gfCNCPoint4[6055] = {X 82.2391, Y 48.2324, Z -5.5000, A 0.000, B 0.000, C 0.000 }
gfCNCPoint4[6056] = {X 81.7221, Y 47.5300, Z -5.5000, A 0.000, B 0.000, C 0.000 }
gfCNCPoint4[6057] = {X 81.3384, Y 46.7467, Z -5.5000, A 0.000, B 0.000, C 0.000 }
gfCNCPoint4[6058] = {X 81.1002, Y 45.9077, Z -5.5000, A 0.000, B 0.000, C 0.000 }
gfCNCPoint4[6059] = {X 81.0152, Y 45.0397, Z -5.5000, A 0.000, B 0.000, C 0.000 }
gfCNCPoint4[6060] = {X 81.0151, Y 44.2040, Z -5.5000, A 0.000, B 0.000, C 0.000 }
gfCNCPoint4[6061] = {X 81.1197, Y 43.2202, Z -5.5000, A 0.000, B 0.000, C 0.000 }
gfCNCPoint4[6062] = {X 81.4183, Y 42.2769, Z -5.5000, A 0.000, B 0.000, C 0.000 }
gfCNCPoint4[6063] = {X 81.8990, Y 41.4122, Z -5.5000, A 0.000, B 0.000, C 0.000 }
gfCNCPoint4[6064] = {X 82.5425, Y 40.6607, Z -5.5000, A 0.000, B 0.000, C 0.000 }
gfCNCPoint4[6065] = {X 82.5423, Y 25.2486, Z -5.5000, A 0.000, B 0.000, C 0.000 }
gfCNCPoint4[6066] = {X 77.7423, Y 25.2486, Z -5.5000, A 0.000, B 0.000, C 0.000 }
gfCNCPoint4[6067] = {X 77.7422, Y 18.1966, Z -5.5000, A 0.000, B 0.000, C 0.000 }
gfCNCPoint4[6068] = {X 77.0779, Y 16.9730, Z -5.5000, A 0.000, B 0.000, C 0.000 }
gfCNCPoint4[6069] = {X 76.5960, Y 15.6668, Z -5.5000, A 0.000, B 0.000, C 0.000 }
gfCNCPoint4[6070] = {X 76.3064, Y 14.3049, Z -5.5000, A 0.000, B 0.000, C 0.000 }
gfCNCPoint4[6071] = {X 74.0412, Y 14.3049, Z -5.5000, A 0.000, B 0.000, C 0.000 }
gfCNCPoint4[6072] = {X 73.9993, Y 14.7005, Z -5.5000, A 0.000, B 0.000, C 0.000 }
gfCNCPoint4[6073] = {X 73.9466, Y 15.0949, Z -5.5000, A 0.000, B 0.000, C 0.000 }
gfCNCPoint4[6074] = {X 77.7423, Y 25.2486, Z -5.5000, A 0.000, B 0.000, C 0.000 }
gfCNCPoint4[6075] = {X 80.1423, Y 25.2486, Z -5.5000, A 0.000, B 0.000, C 0.000 }
gfCNCPoint4[6076] = {X 80.1422, Y 17.4393, Z -5.5000, A 0.000, B 0.000, C 0.000 }
gfCNCPoint4[6077] = {X 79.4941, Y 16.4459, Z -5.5000, A 0.000, B 0.000, C 0.000 }
gfCNCPoint4[6078] = {X 79.0159, Y 15.3604, Z -5.5000, A 0.000, B 0.000, C 0.000 }
gfCNCPoint4[6079] = {X 78.7203, Y 14.2116, Z -5.5000, A 0.000, B 0.000, C 0.000 }
gfCNCPoint4[6080] = {X 78.6153, Y 13.0301, Z -5.5000, A 0.000, B 0.000, C 0.000 }
gfCNCPoint4[6081] = {X 78.6151, Y 12.1868, Z -5.5000, A 0.000, B 0.000, C 0.000 }
gfCNCPoint4[6082] = {X 78.6164, Y 12.0458, Z -5.5000, A 0.000, B 0.000, C 0.000 }
gfCNCPoint4[6083] = {X 78.6205, Y 11.9049, Z -5.5000, A 0.000, B 0.000, C 0.000 }
gfCNCPoint4[6084] = {X 71.6988, Y 11.9049, Z -5.5000, A 0.000, B 0.000, C 0.000 }
gfCNCPoint4[6085] = {X 71.7013, Y 12.0459, Z -5.5000, A 0.000, B 0.000, C 0.000 }
gfCNCPoint4[6086] = {X 71.7021, Y 12.1868, Z -5.5000, A 0.000, B 0.000, C 0.000 }
gfCNCPoint4[6087] = {X 71.7016, Y 13.0911, Z -5.5000, A 0.000, B 0.000, C 0.000 }
gfCNCPoint4[6088] = {X 71.6386, Y 14.2148, Z -5.5000, A 0.000, B 0.000, C 0.000 }
gfCNCPoint4[6089] = {X 71.4714, Y 15.3277, Z -5.5000, A 0.000, B 0.000, C 0.000 }
gfCNCPoint4[6090] = {X 78.9558, Y 35.3487, Z -5.5000, A 0.000, B 0.000, C 0.000 }
gfCNCPoint4[6091] = {X 79.5720, Y 35.9625, Z -5.5000, A 0.000, B 0.000, C 0.000 }
gfCNCPoint4[6092] = {X 80.1424, Y 36.6190, Z -5.5000, A 0.000, B 0.000, C 0.000 }
gfCNCPoint4[6093] = {X 80.1423, Y 25.2486, Z -5.5000, A 0.000, B 0.000, C 0.000 }
gfCNCPoint4[6094] = {X 82.5423, Y 25.2486, Z -5.5000, A 0.000, B 0.000, C 0.000 }
gfCNCPoint4[6095] = {X 82.5422, Y 16.5238, Z -5.5000, A 0.000, B 0.000, C 0.000 }
gfCNCPoint4[6096] = {X 81.9012, Y 15.7822, Z -5.5000, A 0.000, B 0.000, C 0.000 }
gfCNCPoint4[6097] = {X 81.4214, Y 14.9274, Z -5.5000, A 0.000, B 0.000, C 0.000 }
gfCNCPoint4[6098] = {X 81.1220, Y 13.9940, Z -5.5000, A 0.000, B 0.000, C 0.000 }
gfCNCPoint4[6099] = {X 81.0153, Y 13.0196, Z -5.5000, A 0.000, B 0.000, C 0.000 }
gfCNCPoint4[6100] = {X 81.0151, Y 12.1868, Z -5.5000, A 0.000, B 0.000, C 0.000 }
gfCNCPoint4[6101] = {X 81.0160, Y 12.0923, Z -5.5000, A 0.000, B 0.000, C 0.000 }
gfCNCPoint4[6102] = {X 81.0187, Y 11.9979, Z -5.5000, A 0.000, B 0.000, C 0.000 }
gfCNCPoint4[6103] = {X 81.1324, Y 11.1230, Z -5.5000, A 0.000, B 0.000, C 0.000 }
gfCNCPoint4[6104] = {X 81.4018, Y 10.2828, Z -5.5000, A 0.000, B 0.000, C 0.000 }
gfCNCPoint4[6105] = {X 81.8181, Y 9.5049, Z -5.5000, A 0.000, B 0.000, C 0.000 }
gfCNCPoint4[6106] = {X 82.2191, Y 9.7687, Z -5.5000, A 0.000, B 0.000, C 0.000 }
gfCNCPoint4[6107] = {X 82.7659, Y 9.0935, Z -5.5000, A 0.000, B 0.000, C 0.000 }
gfCNCPoint4[6108] = {X 83.4348, Y 8.5389, Z -5.5000, A 0.000, B 0.000, C 0.000 }
gfCNCPoint4[6109] = {X 84.1996, Y 8.1266, Z -5.5000, A 0.000, B 0.000, C 0.000 }
gfCNCPoint4[6110] = {X 85.0305, Y 7.8726, Z -5.5000, A 0.000, B 0.000, C 0.000 }
gfCNCPoint4[6111] = {X 85.8951, Y 7.7868, Z -5.5000, A 0.000, B 0.000, C 0.000 }
gfCNCPoint4[6112] = {X 94.0497, Y 7.7868, Z -5.5000, A 0.000, B 0.000, C 0.000 }
gfCNCPoint4[6113] = {X 95.0288, Y 7.8971, Z -5.5000, A 0.000, B 0.000, C 0.000 }
gfCNCPoint4[6114] = {X 95.9588, Y 8.2226, Z -5.5000, A 0.000, B 0.000, C 0.000 }
gfCNCPoint4[6115] = {X 96.7930, Y 8.7468, Z -5.5000, A 0.000, B 0.000, C 0.000 }
gfCNCPoint4[6116] = {X 97.4897, Y 9.4435, Z -5.5000, A 0.000, B 0.000, C 0.000 }
gfCNCPoint4[6117] = {X 98.0139, Y 10.2777, Z -5.5000, A 0.000, B 0.000, C 0.000 }
gfCNCPoint4[6118] = {X 98.3394, Y 11.2077, Z -5.5000, A 0.000, B 0.000, C 0.000 }
gfCNCPoint4[6119] = {X 98.4497, Y 12.1868, Z -5.5000, A 0.000, B 0.000, C 0.000 }
gfCNCPoint4[6120] = {X 98.4494, Y 13.0233, Z -5.5000, A 0.000, B 0.000, C 0.000 }
gfCNCPoint4[6121] = {X 98.3724, Y 13.7990, Z -5.5000, A 0.000, B 0.000, C 0.000 }
gfCNCPoint4[6122] = {X 98.1597, Y 14.5489, Z -5.5000, A 0.000, B 0.000, C 0.000 }
gfCNCPoint4[6123] = {X 97.8180, Y 15.2496, Z -5.5000, A 0.000, B 0.000, C 0.000 }
gfCNCPoint4[6124] = {X 98.3682, Y 16.6194, Z -5.5000, A 0.000, B 0.000, C 0.000 }
gfCNCPoint4[6125] = {X 101.8748, Y 25.3115, Z -5.5000, A 0.000, B 0.000, C 0.000 }
gfCNCPoint4[6126] = {X 103.4202, Y 21.4659, Z -5.5000, A 0.000, B 0.000, C 0.000 }
gfCNCPoint4[6127] = {X 105.9238, Y 15.2225, Z -5.5000, A 0.000, B 0.000, C 0.000 }
gfCNCPoint4[6128] = {X 105.5855, Y 14.5151, Z -5.5000, A 0.000, B 0.000, C 0.000 }
gfCNCPoint4[6129] = {X 105.3781, Y 13.7589, Z -5.5000, A 0.000, B 0.000, C 0.000 }
gfCNCPoint4[6130] = {X 105.3083, Y 12.9779, Z -5.5000, A 0.000, B 0.000, C 0.000 }
gfCNCPoint4[6131] = {X 105.3083, Y 12.1868, Z -5.5000, A 0.000, B 0.000, C 0.000 }
gfCNCPoint4[6132] = {X 105.4186, Y 11.2077, Z -5.5000, A 0.000, B 0.000, C 0.000 }
gfCNCPoint4[6133] = {X 105.7440, Y 10.2777, Z -5.5000, A 0.000, B 0.000, C 0.000 }
gfCNCPoint4[6134] = {X 106.2682, Y 9.4435, Z -5.5000, A 0.000, B 0.000, C 0.000 }
gfCNCPoint4[6135] = {X 106.9649, Y 8.7468, Z -5.5000, A 0.000, B 0.000, C 0.000 }
gfCNCPoint4[6136] = {X 107.7992, Y 8.2226, Z -5.5000, A 0.000, B 0.000, C 0.000 }
gfCNCPoint4[6137] = {X 108.7292, Y 7.8971, Z -5.5000, A 0.000, B 0.000, C 0.000 }
gfCNCPoint4[6138] = {X 109.7083, Y 7.7868, Z -5.5000, A 0.000, B 0.000, C 0.000 }
gfCNCPoint4[6139] = {X 117.7916, Y 7.7868, Z -5.5000, A 0.000, B 0.000, C 0.000 }
gfCNCPoint4[6140] = {X 118.7707, Y 7.8971, Z -5.5000, A 0.000, B 0.000, C 0.000 }
gfCNCPoint4[6141] = {X 119.7007, Y 8.2226, Z -5.5000, A 0.000, B 0.000, C 0.000 }
gfCNCPoint4[6142] = {X 120.5349, Y 8.7468, Z -5.5000, A 0.000, B 0.000, C 0.000 }
gfCNCPoint4[6143] = {X 121.2316, Y 9.4435, Z -5.5000, A 0.000, B 0.000, C 0.000 }
gfCNCPoint4[6144] = {X 121.7558, Y 10.2777, Z -5.5000, A 0.000, B 0.000, C 0.000 }
gfCNCPoint4[6145] = {X 122.0813, Y 11.2077, Z -5.5000, A 0.000, B 0.000, C 0.000 }
gfCNCPoint4[6146] = {X 122.1916, Y 12.1868, Z -5.5000, A 0.000, B 0.000, C 0.000 }
gfCNCPoint4[6147] = {X 122.1913, Y 13.0233, Z -5.5000, A 0.000, B 0.000, C 0.000 }
gfCNCPoint4[6148] = {X 122.0831, Y 13.9490, Z -5.5000, A 0.000, B 0.000, C 0.000 }
gfCNCPoint4[6149] = {X 121.7823, Y 14.8311, Z -5.5000, A 0.000, B 0.000, C 0.000 }
gfCNCPoint4[6150] = {X 121.3025, Y 15.6301, Z -5.5000, A 0.000, B 0.000, C 0.000 }
gfCNCPoint4[6151] = {X 120.6651, Y 16.3101, Z -5.5000, A 0.000, B 0.000, C 0.000 }
gfCNCPoint4[6152] = {X 120.6644, Y 40.8765, Z -5.5000, A 0.000, B 0.000, C 0.000 }
gfCNCPoint4[6153] = {X 120.6784, Y 40.8882, Z -5.5000, A 0.000, B 0.000, C 0.000 }
gfCNCPoint4[6154] = {X 121.3172, Y 41.5763, Z -5.5000, A 0.000, B 0.000, C 0.000 }
gfCNCPoint4[6155] = {X 121.7955, Y 42.3843, Z -5.5000, A 0.000, B 0.000, C 0.000 }
gfCNCPoint4[6156] = {X 122.0914, Y 43.2753, Z -5.5000, A 0.000, B 0.000, C 0.000 }
gfCNCPoint4[6157] = {X 122.1916, Y 44.2089, Z -5.5000, A 0.000, B 0.000, C 0.000 }
gfCNCPoint4[6158] = {X 122.1916, Y 45.0000, Z -5.5000, A 0.000, B 0.000, C 0.000 }
gfCNCPoint4[6159] = {X 122.0813, Y 45.9791, Z -5.5000, A 0.000, B 0.000, C 0.000 }
gfCNCPoint4[6160] = {X 121.7558, Y 46.9091, Z -5.5000, A 0.000, B 0.000, C 0.000 }
gfCNCPoint4[6161] = {X 121.2316, Y 47.7434, Z -5.5000, A 0.000, B 0.000, C 0.000 }
gfCNCPoint4[6162] = {X 120.5349, Y 48.4401, Z -5.5000, A 0.000, B 0.000, C 0.000 }
gfCNCPoint4[6163] = {X 119.7007, Y 48.9643, Z -5.5000, A 0.000, B 0.000, C 0.000 }
gfCNCPoint4[6164] = {X 118.7707, Y 49.2897, Z -5.5000, A 0.000, B 0.000, C 0.000 }
gfCNCPoint4[6165] = {X 117.7916, Y 49.4000, Z -5.5000, A 0.000, B 0.000, C 0.000 }
gfCNCPoint4[6166] = {X 111.9185, Y 49.4000, Z -5.5000, A 0.000, B 0.000, C 0.000 }
gfCNCPoint4[6167] = {X 110.9394, Y 49.2897, Z -5.5000, A 0.000, B 0.000, C 0.000 }
gfCNCPoint4[6168] = {X 110.0094, Y 48.9643, Z -5.5000, A 0.000, B 0.000, C 0.000 }
gfCNCPoint4[6169] = {X 109.1751, Y 48.4400, Z -5.5000, A 0.000, B 0.000, C 0.000 }
gfCNCPoint4[6170] = {X 108.4784, Y 47.7433, Z -5.5000, A 0.000, B 0.000, C 0.000 }
gfCNCPoint4[6171] = {X 107.9542, Y 46.9091, Z -5.5000, A 0.000, B 0.000, C 0.000 }
gfCNCPoint4[6172] = {X 107.6288, Y 45.9791, Z -5.5000, A 0.000, B 0.000, C 0.000 }
gfCNCPoint4[6173] = {X 107.5185, Y 45.0000, Z -5.5000, A 0.000, B 0.000, C 0.000 }
gfCNCPoint4[6174] = {X 107.5185, Y 44.1807, Z -5.5000, A 0.000, B 0.000, C 0.000 }
gfCNCPoint4[6175] = {X 107.5549, Y 43.6258, Z -5.5000, A 0.000, B 0.000, C 0.000 }
gfCNCPoint4[6176] = {X 107.6637, Y 43.0805, Z -5.5000, A 0.000, B 0.000, C 0.000 }
gfCNCPoint4[6177] = {X 106.1856, Y 46.6923, Z -5.5000, A 0.000, B 0.000, C 0.000 }
gfCNCPoint4[6178] = {X 105.8087, Y 47.4049, Z -5.5000, A 0.000, B 0.000, C 0.000 }
gfCNCPoint4[6179] = {X 105.3081, Y 48.0367, Z -5.5000, A 0.000, B 0.000, C 0.000 }
gfCNCPoint4[6180] = {X 104.7006, Y 48.5667, Z -5.5000, A 0.000, B 0.000, C 0.000 }
gfCNCPoint4[6181] = {X 104.0067, Y 48.9769, Z -5.5000, A 0.000, B 0.000, C 0.000 }
gfCNCPoint4[6182] = {X 103.0414, Y 49.3033, Z -5.5000, A 0.000, B 0.000, C 0.000 }
gfCNCPoint4[6183] = {X 102.0269, Y 49.3989, Z -5.5000, A 0.000, B 0.000, C 0.000 }
gfCNCPoint4[6184] = {X 101.0176, Y 49.2586, Z -5.5000, A 0.000, B 0.000, C 0.000 }
gfCNCPoint4[6185] = {X 100.0676, Y 48.8899, Z -5.5000, A 0.000, B 0.000, C 0.000 }
gfCNCPoint4[6186] = {X 99.2280, Y 48.3125, Z -5.5000, A 0.000, B 0.000, C 0.000 }
gfCNCPoint4[6187] = {X 98.5436, Y 47.5575, Z -5.5000, A 0.000, B 0.000, C 0.000 }
gfCNCPoint4[6188] = {X 98.0514, Y 46.6653, Z -5.5000, A 0.000, B 0.000, C 0.000 }
gfCNCPoint4[6189] = {X 96.5880, Y 43.0864, Z -5.5000, A 0.000, B 0.000, C 0.000 }
gfCNCPoint4[6190] = {X 96.6989, Y 43.6428, Z -5.5000, A 0.000, B 0.000, C 0.000 }
gfCNCPoint4[6191] = {X 96.7385, Y 44.2089, Z -5.5000, A 0.000, B 0.000, C 0.000 }
gfCNCPoint4[6192] = {X 96.7383, Y 45.0423, Z -5.5000, A 0.000, B 0.000, C 0.000 }
gfCNCPoint4[6193] = {X 96.6200, Y 46.0144, Z -5.5000, A 0.000, B 0.000, C 0.000 }
gfCNCPoint4[6194] = {X 96.2896, Y 46.9363, Z -5.5000, A 0.000, B 0.000, C 0.000 }
gfCNCPoint4[6195] = {X 95.7635, Y 47.7622, Z -5.5000, A 0.000, B 0.000, C 0.000 }
gfCNCPoint4[6196] = {X 95.0677, Y 48.4513, Z -5.5000, A 0.000, B 0.000, C 0.000 }
gfCNCPoint4[6197] = {X 94.2367, Y 48.9695, Z -5.5000, A 0.000, B 0.000, C 0.000 }
gfCNCPoint4[6198] = {X 93.3117, Y 49.2910, Z -5.5000, A 0.000, B 0.000, C 0.000 }
gfCNCPoint4[6199] = {X 92.3385, Y 49.4000, Z -5.5000, A 0.000, B 0.000, C 0.000 }
gfCNCPoint4[6200] = {X 85.8951, Y 49.4000, Z -5.5000, A 0.000, B 0.000, C 0.000 }
gfCNCPoint4[6201] = {X 84.9160, Y 49.2897, Z -5.5000, A 0.000, B 0.000, C 0.000 }
gfCNCPoint4[6202] = {X 83.9860, Y 48.9643, Z -5.5000, A 0.000, B 0.000, C 0.000 }
gfCNCPoint4[6203] = {X 83.1517, Y 48.4400, Z -5.5000, A 0.000, B 0.000, C 0.000 }
gfCNCPoint4[6204] = {X 82.4550, Y 47.7433, Z -5.5000, A 0.000, B 0.000, C 0.000 }
gfCNCPoint4[6205] = {X 81.9308, Y 46.9091, Z -5.5000, A 0.000, B 0.000, C 0.000 }
gfCNCPoint4[6206] = {X 81.6054, Y 45.9791, Z -5.5000, A 0.000, B 0.000, C 0.000 }
gfCNCPoint4[6207] = {X 81.4951, Y 45.0000, Z -5.5000, A 0.000, B 0.000, C 0.000 }
gfCNCPoint4[6208] = {X 81.4951, Y 44.2067, Z -5.5000, A 0.000, B 0.000, C 0.000 }
gfCNCPoint4[6209] = {X 81.6001, Y 43.2693, Z -5.5000, A 0.000, B 0.000, C 0.000 }
gfCNCPoint4[6210] = {X 81.8999, Y 42.3751, Z -5.5000, A 0.000, B 0.000, C 0.000 }
gfCNCPoint4[6211] = {X 82.3813, Y 41.5640, Z -5.5000, A 0.000, B 0.000, C 0.000 }
gfCNCPoint4[6212] = {X 83.0225, Y 40.8723, Z -5.5000, A 0.000, B 0.000, C 0.000 }
gfCNCPoint4[6213] = {X 83.0222, Y 16.3107, Z -5.5000, A 0.000, B 0.000, C 0.000 }
gfCNCPoint4[6214] = {X 82.3778, Y 15.6216, Z -5.5000, A 0.000, B 0.000, C 0.000 }
gfCNCPoint4[6215] = {X 81.8950, Y 14.8109, Z -5.5000, A 0.000, B 0.000, C 0.000 }
gfCNCPoint4[6216] = {X 81.5962, Y 13.9160, Z -5.5000, A 0.000, B 0.000, C 0.000 }
gfCNCPoint4[6217] = {X 81.4951, Y 12.9780, Z -5.5000, A 0.000, B 0.000, C 0.000 }
gfCNCPoint4[6218] = {X 81.4951, Y 12.1868, Z -5.5000, A 0.000, B 0.000, C 0.000 }
gfCNCPoint4[6219] = {X 81.5776, Y 11.3388, Z -5.5000, A 0.000, B 0.000, C 0.000 }
gfCNCPoint4[6220] = {X 81.8220, Y 10.5226, Z -5.5000, A 0.000, B 0.000, C 0.000 }
gfCNCPoint4[6221] = {X 82.2191, Y 9.7687, Z -5.5000, A 0.000, B 0.000, C 0.000 }
gfCNCPoint4[6222] = {X 81.8181, Y 9.5049, Z -5.5000, A 0.000, B 0.000, C 0.000 }
gfCNCPoint4[6223] = {X 68.9232, Y 9.5049, Z -5.5000, A 0.000, B 0.000, C 0.000 }
gfCNCPoint4[6224] = {X 69.1905, Y 10.7208, Z -5.5000, A 0.000, B 0.000, C 0.000 }
gfCNCPoint4[6225] = {X 69.2995, Y 11.9609, Z -5.5000, A 0.000, B 0.000, C 0.000 }
gfCNCPoint4[6226] = {X 69.3015, Y 12.0739, Z -5.5000, A 0.000, B 0.000, C 0.000 }
gfCNCPoint4[6227] = {X 69.3021, Y 12.1868, Z -5.5000, A 0.000, B 0.000, C 0.000 }
gfCNCPoint4[6228] = {X 69.3017, Y 13.0687, Z -5.5000, A 0.000, B 0.000, C 0.000 }
gfCNCPoint4[6229] = {X 69.2127, Y 14.2904, Z -5.5000, A 0.000, B 0.000, C 0.000 }
gfCNCPoint4[6230] = {X 68.9702, Y 15.4910, Z -5.5000, A 0.000, B 0.000, C 0.000 }
gfCNCPoint4[6231] = {X 76.9187, Y 36.7535, Z -5.5000, A 0.000, B 0.000, C 0.000 }
gfCNCPoint4[6232] = {X 77.6313, Y 37.4063, Z -5.5000, A 0.000, B 0.000, C 0.000 }
gfCNCPoint4[6233] = {X 78.2753, Y 38.1269, Z -5.5000, A 0.000, B 0.000, C 0.000 }
gfCNCPoint4[6234] = {X 79.0229, Y 39.1918, Z -5.5000, A 0.000, B 0.000, C 0.000 }
gfCNCPoint4[6235] = {X 79.6209, Y 40.3474, Z -5.5000, A 0.000, B 0.000, C 0.000 }
gfCNCPoint4[6236] = {X 80.0586, Y 41.5727, Z -5.5000, A 0.000, B 0.000, C 0.000 }
gfCNCPoint4[6237] = {X 80.3280, Y 42.8456, Z -5.5000, A 0.000, B 0.000, C 0.000 }
gfCNCPoint4[6238] = {X 80.4242, Y 44.1432, Z -5.5000, A 0.000, B 0.000, C 0.000 }
gfCNCPoint4[6239] = {X 80.4245, Y 45.0000, Z -5.5000, A 0.000, B 0.000, C 0.000 }
gfCNCPoint4[6240] = {X 80.3511, Y 46.1898, Z -5.5000, A 0.000, B 0.000, C 0.000 }
gfCNCPoint4[6241] = {X 80.1320, Y 47.3615, Z -5.5000, A 0.000, B 0.000, C 0.000 }
gfCNCPoint4[6242] = {X 79.7706, Y 48.4974, Z -5.5000, A 0.000, B 0.000, C 0.000 }
gfCNCPoint4[6243] = {X 79.2722, Y 49.5803, Z -5.5000, A 0.000, B 0.000, C 0.000 }
gfCNCPoint4[6244] = {X 78.4688, Y 50.8341, Z -5.5000, A 0.000, B 0.000, C 0.000 }
gfCNCPoint4[6245] = {X 77.4826, Y 51.9498, Z -5.5000, A 0.000, B 0.000, C 0.000 }
gfCNCPoint4[6246] = {X 76.3369, Y 52.9011, Z -5.5000, A 0.000, B 0.000, C 0.000 }
gfCNCPoint4[6247] = {X 75.0589, Y 53.6653, Z -5.5000, A 0.000, B 0.000, C 0.000 }
gfCNCPoint4[6248] = {X 73.6787, Y 54.2246, Z -5.5000, A 0.000, B 0.000, C 0.000 }
gfCNCPoint4[6249] = {X 72.2292, Y 54.5655, Z -5.5000, A 0.000, B 0.000, C 0.000 }
gfCNCPoint4[6250] = {X 70.7445, Y 54.6800, Z -5.5000, A 0.000, B 0.000, C 0.000 }
gfCNCPoint4[6251] = {X 64.1851, Y 54.6800, Z -5.5000, A 0.000, B 0.000, C 0.000 }
gfCNCPoint4[6252] = {X 62.7229, Y 54.5689, Z -5.5000, A 0.000, B 0.000, C 0.000 }
gfCNCPoint4[6253] = {X 61.2943, Y 54.2383, Z -5.5000, A 0.000, B 0.000, C 0.000 }
gfCNCPoint4[6254] = {X 59.9320, Y 53.6956, Z -5.5000, A 0.000, B 0.000, C 0.000 }
gfCNCPoint4[6255] = {X 58.6673, Y 52.9534, Z -5.5000, A 0.000, B 0.000, C 0.000 }
gfCNCPoint4[6256] = {X 57.5293, Y 52.0286, Z -5.5000, A 0.000, B 0.000, C 0.000 }
gfCNCPoint4[6257] = {X 56.6337, Y 51.0563, Z -5.5000, A 0.000, B 0.000, C 0.000 }
gfCNCPoint4[6258] = {X 55.8790, Y 49.9710, Z -5.5000, A 0.000, B 0.000, C 0.000 }
gfCNCPoint4[6259] = {X 55.1243, Y 51.0563, Z -5.5000, A 0.000, B 0.000, C 0.000 }
gfCNCPoint4[6260] = {X 54.2288, Y 52.0286, Z -5.5000, A 0.000, B 0.000, C 0.000 }
gfCNCPoint4[6261] = {X 53.0907, Y 52.9534, Z -5.5000, A 0.000, B 0.000, C 0.000 }
gfCNCPoint4[6262] = {X 51.8261, Y 53.6956, Z -5.5000, A 0.000, B 0.000, C 0.000 }
gfCNCPoint4[6263] = {X 50.4638, Y 54.2383, Z -5.5000, A 0.000, B 0.000, C 0.000 }
gfCNCPoint4[6264] = {X 49.0351, Y 54.5689, Z -5.5000, A 0.000, B 0.000, C 0.000 }
gfCNCPoint4[6265] = {X 47.5729, Y 54.6800, Z -5.5000, A 0.000, B 0.000, C 0.000 }
gfCNCPoint4[6266] = {X 40.6393, Y 54.6800, Z -5.5000, A 0.000, B 0.000, C 0.000 }
gfCNCPoint4[6267] = {X 39.2448, Y 54.5790, Z -5.5000, A 0.000, B 0.000, C 0.000 }
gfCNCPoint4[6268] = {X 37.8793, Y 54.2782, Z -5.5000, A 0.000, B 0.000, C 0.000 }
gfCNCPoint4[6269] = {X 36.5715, Y 53.7838, Z -5.5000, A 0.000, B 0.000, C 0.000 }
gfCNCPoint4[6270] = {X 35.3485, Y 53.1062, Z -5.5000, A 0.000, B 0.000, C 0.000 }
gfCNCPoint4[6271] = {X 33.9153, Y 54.1346, Z -5.5000, A 0.000, B 0.000, C 0.000 }
gfCNCPoint4[6272] = {X 32.3642, Y 54.9748, Z -5.5000, A 0.000, B 0.000, C 0.000 }
gfCNCPoint4[6273] = {X 30.7198, Y 55.6135, Z -5.5000, A 0.000, B 0.000, C 0.000 }
gfCNCPoint4[6274] = {X 29.0082, Y 56.0405, Z -5.5000, A 0.000, B 0.000, C 0.000 }
gfCNCPoint4[6275] = {X 27.2565, Y 56.2491, Z -5.5000, A 0.000, B 0.000, C 0.000 }
gfCNCPoint4[6276] = {X 24.9813, Y 57.2329, Z -5.5000, A 0.000, B 0.000, C 0.000 }
gfCNCPoint4[6277] = {X 22.6481, Y 58.0696, Z -5.5000, A 0.000, B 0.000, C 0.000 }
gfCNCPoint4[6278] = {X 20.0860, Y 58.7984, Z -5.5000, A 0.000, B 0.000, C 0.000 }
gfCNCPoint4[6279] = {X 17.4728, Y 59.3146, Z -5.5000, A 0.000, B 0.000, C 0.000 }
gfCNCPoint4[6280] = {X 14.8260, Y 59.6146, Z -5.5000, A 0.000, B 0.000, C 0.000 }
gfCNCPoint4[6281] = {X 12.1636, Y 59.6965, Z -5.5000, A 0.000, B 0.000, C 0.000 }
gfCNCPoint4[6282] = {X 9.5034, Y 59.5598, Z -5.5000, A 0.000, B 0.000, C 0.000 }
gfCNCPoint4[6283] = {X 9.5034, Y 90.4951, Z -5.5000, A 0.000, B 0.000, C 0.000 }
gfCNCPoint4[6284] = {X 114.8628, Y 90.4951, Z -5.5000, A 0.000, B 0.000, C 0.000 }
gfCNCPoint4[6285] = {X 115.7472, Y 89.2982, Z -5.5000, A 0.000, B 0.000, C 0.000 }
gfCNCPoint4[6286] = {X 116.7720, Y 88.2192, Z -5.5000, A 0.000, B 0.000, C 0.000 }
gfCNCPoint4[6287] = {X 117.9218, Y 87.2744, Z -5.5000, A 0.000, B 0.000, C 0.000 }
gfCNCPoint4[6288] = {X 119.1789, Y 86.4781, Z -5.5000, A 0.000, B 0.000, C 0.000 }
gfCNCPoint4[6289] = {X 120.5245, Y 85.8425, Z -5.5000, A 0.000, B 0.000, C 0.000 }
gfCNCPoint4[6290] = {X 121.9380, Y 85.3771, Z -5.5000, A 0.000, B 0.000, C 0.000 }
gfCNCPoint4[6291] = {X 123.3980, Y 85.0890, Z -5.5000, A 0.000, B 0.000, C 0.000 }
gfCNCPoint4[6292] = {X 123.5627, Y 84.9116, Z -5.5000, A 0.000, B 0.000, C 0.000 }
gfCNCPoint4[6293] = {X 123.7255, Y 84.7325, Z -5.5000, A 0.000, B 0.000, C 0.000 }
gfCNCPoint4[6294] = {X 147.2181, Y 58.9343, Z -5.5000, A 0.000, B 0.000, C 0.000 }
gfCNCPoint4[6295] = {X 147.2180, Y 58.0000, Z -5.5000, A 0.000, B 0.000, C 0.000 }
gfCNCPoint4[6296] = {X 147.2987, Y 56.6058, Z -5.5000, A 0.000, B 0.000, C 0.000 }
gfCNCPoint4[6297] = {X 147.5398, Y 55.2303, Z -5.5000, A 0.000, B 0.000, C 0.000 }
gfCNCPoint4[6298] = {X 148.0022, Y 53.7185, Z -5.5000, A 0.000, B 0.000, C 0.000 }
gfCNCPoint4[6299] = {X 148.6580, Y 52.2800, Z -5.5000, A 0.000, B 0.000, C 0.000 }
gfCNCPoint4[6300] = {X 143.0396, Y 52.2800, Z -5.5000, A 0.000, B 0.000, C 0.000 }
gfCNCPoint4[6301] = {X 141.7807, Y 52.1703, Z -5.5000, A 0.000, B 0.000, C 0.000 }
gfCNCPoint4[6302] = {X 140.5597, Y 51.8446, Z -5.5000, A 0.000, B 0.000, C 0.000 }
gfCNCPoint4[6303] = {X 139.4134, Y 51.3126, Z -5.5000, A 0.000, B 0.000, C 0.000 }
gfCNCPoint4[6304] = {X 138.3764, Y 50.5904, Z -5.5000, A 0.000, B 0.000, C 0.000 }
gfCNCPoint4[6305] = {X 137.4799, Y 49.6998, Z -5.5000, A 0.000, B 0.000, C 0.000 }
gfCNCPoint4[6306] = {X 136.7509, Y 48.6675, Z -5.5000, A 0.000, B 0.000, C 0.000 }
gfCNCPoint4[6307] = {X 136.2114, Y 47.5248, Z -5.5000, A 0.000, B 0.000, C 0.000 }
gfCNCPoint4[6308] = {X 135.8777, Y 46.3059, Z -5.5000, A 0.000, B 0.000, C 0.000 }
gfCNCPoint4[6309] = {X 135.7598, Y 45.0477, Z -5.5000, A 0.000, B 0.000, C 0.000 }
gfCNCPoint4[6310] = {X 135.7601, Y 44.1248, Z -5.5000, A 0.000, B 0.000, C 0.000 }
gfCNCPoint4[6311] = {X 135.8408, Y 43.1249, Z -5.5000, A 0.000, B 0.000, C 0.000 }
gfCNCPoint4[6312] = {X 136.0581, Y 42.1457, Z -5.5000, A 0.000, B 0.000, C 0.000 }
gfCNCPoint4[6313] = {X 138.3597, Y 42.8258, Z -5.5000, A 0.000, B 0.000, C 0.000 }
gfCNCPoint4[6314] = {X 138.6721, Y 42.0319, Z -5.5000, A 0.000, B 0.000, C 0.000 }
gfCNCPoint4[6315] = {X 139.1179, Y 41.3046, Z -5.5000, A 0.000, B 0.000, C 0.000 }
gfCNCPoint4[6316] = {X 139.6836, Y 40.6660, Z -5.5000, A 0.000, B 0.000, C 0.000 }
gfCNCPoint4[6317] = {X 139.6836, Y 20.4376, Z -5.5000, A 0.000, B 0.000, C 0.000 }
gfCNCPoint4[6318] = {X 137.7100, Y 20.4373, Z -5.5000, A 0.000, B 0.000, C 0.000 }
gfCNCPoint4[6319] = {X 136.9998, Y 21.1824, Z -5.5000, A 0.000, B 0.000, C 0.000 }
gfCNCPoint4[6320] = {X 136.1491, Y 21.7619, Z -5.5000, A 0.000, B 0.000, C 0.000 }
gfCNCPoint4[6321] = {X 135.4282, Y 22.0767, Z -5.5000, A 0.000, B 0.000, C 0.000 }
gfCNCPoint4[6322] = {X 134.6660, Y 22.2715, Z -5.5000, A 0.000, B 0.000, C 0.000 }
gfCNCPoint4[6323] = {X 133.8824, Y 22.3414, Z -5.5000, A 0.000, B 0.000, C 0.000 }
gfCNCPoint4[6324] = {X 133.2006, Y 22.3415, Z -5.5000, A 0.000, B 0.000, C 0.000 }
gfCNCPoint4[6325] = {X 132.2486, Y 22.2478, Z -5.5000, A 0.000, B 0.000, C 0.000 }
gfCNCPoint4[6326] = {X 131.3331, Y 21.9701, Z -5.5000, A 0.000, B 0.000, C 0.000 }
gfCNCPoint4[6327] = {X 130.4895, Y 21.5191, Z -5.5000, A 0.000, B 0.000, C 0.000 }
gfCNCPoint4[6328] = {X 129.7500, Y 20.9122, Z -5.5000, A 0.000, B 0.000, C 0.000 }
gfCNCPoint4[6329] = {X 129.1431, Y 20.1727, Z -5.5000, A 0.000, B 0.000, C 0.000 }
gfCNCPoint4[6330] = {X 128.6921, Y 19.3290, Z -5.5000, A 0.000, B 0.000, C 0.000 }
gfCNCPoint4[6331] = {X 128.4144, Y 18.4136, Z -5.5000, A 0.000, B 0.000, C 0.000 }
gfCNCPoint4[6332] = {X 128.3206, Y 17.4615, Z -5.5000, A 0.000, B 0.000, C 0.000 }
gfCNCPoint4[6333] = {X 128.3206, Y 10.4835, Z -5.5000, A 0.000, B 0.000, C 0.000 }
gfCNCPoint4[6334] = {X 128.3317, Y 10.1548, Z -5.5000, A 0.000, B 0.000, C 0.000 }
gfCNCPoint4[6335] = {X 128.3649, Y 9.8275, Z -5.5000, A 0.000, B 0.000, C 0.000 }
gfCNCPoint4[6336] = {X 128.6079, Y 8.8341, Z -5.5000, A 0.000, B 0.000, C 0.000 }
gfCNCPoint4[6337] = {X 129.0525, Y 7.9131, Z -5.5000, A 0.000, B 0.000, C 0.000 }
gfCNCPoint4[6338] = {X 129.6793, Y 7.1049, Z -5.5000, A 0.000, B 0.000, C 0.000 }
gfCNCPoint4[6339] = {X 130.0257, Y 7.4373, Z -5.5000, A 0.000, B 0.000, C 0.000 }
gfCNCPoint4[6340] = {X 130.6997, Y 6.8634, Z -5.5000, A 0.000, B 0.000, C 0.000 }
gfCNCPoint4[6341] = {X 131.4749, Y 6.4361, Z -5.5000, A 0.000, B 0.000, C 0.000 }
gfCNCPoint4[6342] = {X 132.3200, Y 6.1726, Z -5.5000, A 0.000, B 0.000, C 0.000 }
gfCNCPoint4[6343] = {X 133.2007, Y 6.0835, Z -5.5000, A 0.000, B 0.000, C 0.000 }
gfCNCPoint4[6344] = {X 133.8874, Y 6.0837, Z -5.5000, A 0.000, B 0.000, C 0.000 }
gfCNCPoint4[6345] = {X 134.7188, Y 6.1717, Z -5.5000, A 0.000, B 0.000, C 0.000 }
gfCNCPoint4[6346] = {X 135.5185, Y 6.4153, Z -5.5000, A 0.000, B 0.000, C 0.000 }
gfCNCPoint4[6347] = {X 136.2577, Y 6.8057, Z -5.5000, A 0.000, B 0.000, C 0.000 }
gfCNCPoint4[6348] = {X 136.9097, Y 7.3289, Z -5.5000, A 0.000, B 0.000, C 0.000 }
gfCNCPoint4[6349] = {X 137.4509, Y 7.9660, Z -5.5000, A 0.000, B 0.000, C 0.000 }
gfCNCPoint4[6350] = {X 155.0718, Y 7.9660, Z -5.5000, A 0.000, B 0.000, C 0.000 }
gfCNCPoint4[6351] = {X 155.6196, Y 7.3226, Z -5.5000, A 0.000, B 0.000, C 0.000 }
gfCNCPoint4[6352] = {X 156.2802, Y 6.7958, Z -5.5000, A 0.000, B 0.000, C 0.000 }
gfCNCPoint4[6353] = {X 157.0294, Y 6.4050, Z -5.5000, A 0.000, B 0.000, C 0.000 }
gfCNCPoint4[6354] = {X 157.8395, Y 6.1646, Z -5.5000, A 0.000, B 0.000, C 0.000 }
gfCNCPoint4[6355] = {X 158.6806, Y 6.0835, Z -5.5000, A 0.000, B 0.000, C 0.000 }
gfCNCPoint4[6356] = {X 159.3791, Y 6.0839, Z -5.5000, A 0.000, B 0.000, C 0.000 }
gfCNCPoint4[6357] = {X 160.3488, Y 6.2050, Z -5.5000, A 0.000, B 0.000, C 0.000 }
gfCNCPoint4[6358] = {X 161.2678, Y 6.5371, Z -5.5000, A 0.000, B 0.000, C 0.000 }
gfCNCPoint4[6359] = {X 162.0908, Y 7.0639, Z -5.5000, A 0.000, B 0.000, C 0.000 }
gfCNCPoint4[6360] = {X 162.7773, Y 7.7593, Z -5.5000, A 0.000, B 0.000, C 0.000 }
gfCNCPoint4[6361] = {X 163.2934, Y 8.5891, Z -5.5000, A 0.000, B 0.000, C 0.000 }
gfCNCPoint4[6362] = {X 163.6136, Y 9.5124, Z -5.5000, A 0.000, B 0.000, C 0.000 }
gfCNCPoint4[6363] = {X 163.7221, Y 10.4835, Z -5.5000, A 0.000, B 0.000, C 0.000 }
gfCNCPoint4[6364] = {X 163.7221, Y 17.4615, Z -5.5000, A 0.000, B 0.000, C 0.000 }
gfCNCPoint4[6365] = {X 163.6118, Y 18.4406, Z -5.5000, A 0.000, B 0.000, C 0.000 }
gfCNCPoint4[6366] = {X 163.2863, Y 19.3706, Z -5.5000, A 0.000, B 0.000, C 0.000 }
gfCNCPoint4[6367] = {X 162.7621, Y 20.2049, Z -5.5000, A 0.000, B 0.000, C 0.000 }
gfCNCPoint4[6368] = {X 162.0654, Y 20.9016, Z -5.5000, A 0.000, B 0.000, C 0.000 }
gfCNCPoint4[6369] = {X 161.2312, Y 21.4258, Z -5.5000, A 0.000, B 0.000, C 0.000 }
gfCNCPoint4[6370] = {X 160.3012, Y 21.7512, Z -5.5000, A 0.000, B 0.000, C 0.000 }
gfCNCPoint4[6371] = {X 159.3221, Y 21.8615, Z -5.5000, A 0.000, B 0.000, C 0.000 }
gfCNCPoint4[6372] = {X 158.6789, Y 21.8615, Z -5.5000, A 0.000, B 0.000, C 0.000 }
gfCNCPoint4[6373] = {X 157.8335, Y 21.7768, Z -5.5000, A 0.000, B 0.000, C 0.000 }
gfCNCPoint4[6374] = {X 157.0197, Y 21.5323, Z -5.5000, A 0.000, B 0.000, C 0.000 }
gfCNCPoint4[6375] = {X 156.2676, Y 21.1370, Z -5.5000, A 0.000, B 0.000, C 0.000 }
gfCNCPoint4[6376] = {X 155.6047, Y 20.6055, Z -5.5000, A 0.000, B 0.000, C 0.000 }
gfCNCPoint4[6377] = {X 155.0553, Y 19.9573, Z -5.5000, A 0.000, B 0.000, C 0.000 }
gfCNCPoint4[6378] = {X 152.3567, Y 19.9583, Z -5.5000, A 0.000, B 0.000, C 0.000 }
gfCNCPoint4[6379] = {X 152.3554, Y 40.8428, Z -5.5000, A 0.000, B 0.000, C 0.000 }
gfCNCPoint4[6380] = {X 152.8073, Y 41.3300, Z -5.5000, A 0.000, B 0.000, C 0.000 }
gfCNCPoint4[6381] = {X 152.9004, Y 41.4410, Z -5.5000, A 0.000, B 0.000, C 0.000 }
gfCNCPoint4[6382] = {X 153.4347, Y 42.2813, Z -5.5000, A 0.000, B 0.000, C 0.000 }
gfCNCPoint4[6383] = {X 153.7679, Y 43.2197, Z -5.5000, A 0.000, B 0.000, C 0.000 }
gfCNCPoint4[6384] = {X 153.8831, Y 44.2089, Z -5.5000, A 0.000, B 0.000, C 0.000 }
gfCNCPoint4[6385] = {X 153.8829, Y 45.0423, Z -5.5000, A 0.000, B 0.000, C 0.000 }
gfCNCPoint4[6386] = {X 153.7646, Y 46.0144, Z -5.5000, A 0.000, B 0.000, C 0.000 }
gfCNCPoint4[6387] = {X 153.4342, Y 46.9363, Z -5.5000, A 0.000, B 0.000, C 0.000 }
gfCNCPoint4[6388] = {X 152.9080, Y 47.7622, Z -5.5000, A 0.000, B 0.000, C 0.000 }
gfCNCPoint4[6389] = {X 152.2123, Y 48.4513, Z -5.5000, A 0.000, B 0.000, C 0.000 }
gfCNCPoint4[6390] = {X 151.3813, Y 48.9695, Z -5.5000, A 0.000, B 0.000, C 0.000 }
gfCNCPoint4[6391] = {X 150.4563, Y 49.2910, Z -5.5000, A 0.000, B 0.000, C 0.000 }
gfCNCPoint4[6392] = {X 149.4831, Y 49.4000, Z -5.5000, A 0.000, B 0.000, C 0.000 }
gfCNCPoint4[6393] = {X 143.0396, Y 49.4000, Z -5.5000, A 0.000, B 0.000, C 0.000 }
gfCNCPoint4[6394] = {X 142.0605, Y 49.2897, Z -5.5000, A 0.000, B 0.000, C 0.000 }
gfCNCPoint4[6395] = {X 141.1305, Y 48.9643, Z -5.5000, A 0.000, B 0.000, C 0.000 }
gfCNCPoint4[6396] = {X 140.2963, Y 48.4400, Z -5.5000, A 0.000, B 0.000, C 0.000 }
gfCNCPoint4[6397] = {X 139.5996, Y 47.7433, Z -5.5000, A 0.000, B 0.000, C 0.000 }
gfCNCPoint4[6398] = {X 139.0754, Y 46.9091, Z -5.5000, A 0.000, B 0.000, C 0.000 }
gfCNCPoint4[6399] = {X 138.7499, Y 45.9791, Z -5.5000, A 0.000, B 0.000, C 0.000 }
gfCNCPoint4[6400] = {X 138.6396, Y 45.0000, Z -5.5000, A 0.000, B 0.000, C 0.000 }
gfCNCPoint4[6401] = {X 138.6400, Y 44.1483, Z -5.5000, A 0.000, B 0.000, C 0.000 }
gfCNCPoint4[6402] = {X 138.7505, Y 43.2275, Z -5.5000, A 0.000, B 0.000, C 0.000 }
gfCNCPoint4[6403] = {X 139.0514, Y 42.3503, Z -5.5000, A 0.000, B 0.000, C 0.000 }
gfCNCPoint4[6404] = {X 139.5295, Y 41.5556, Z -5.5000, A 0.000, B 0.000, C 0.000 }
gfCNCPoint4[6405] = {X 140.1636, Y 40.8789, Z -5.5000, A 0.000, B 0.000, C 0.000 }
gfCNCPoint4[6406] = {X 140.1636, Y 19.9577, Z -5.5000, A 0.000, B 0.000, C 0.000 }
gfCNCPoint4[6407] = {X 137.4661, Y 19.9572, Z -5.5000, A 0.000, B 0.000, C 0.000 }
gfCNCPoint4[6408] = {X 136.9184, Y 20.6076, Z -5.5000, A 0.000, B 0.000, C 0.000 }
gfCNCPoint4[6409] = {X 136.2558, Y 21.1405, Z -5.5000, A 0.000, B 0.000, C 0.000 }
gfCNCPoint4[6410] = {X 135.5032, Y 21.5360, Z -5.5000, A 0.000, B 0.000, C 0.000 }
gfCNCPoint4[6411] = {X 134.6885, Y 21.7794, Z -5.5000, A 0.000, B 0.000, C 0.000 }
gfCNCPoint4[6412] = {X 133.8422, Y 21.8615, Z -5.5000, A 0.000, B 0.000, C 0.000 }
gfCNCPoint4[6413] = {X 133.2006, Y 21.8615, Z -5.5000, A 0.000, B 0.000, C 0.000 }
gfCNCPoint4[6414] = {X 132.2215, Y 21.7512, Z -5.5000, A 0.000, B 0.000, C 0.000 }
gfCNCPoint4[6415] = {X 131.2916, Y 21.4258, Z -5.5000, A 0.000, B 0.000, C 0.000 }
gfCNCPoint4[6416] = {X 130.4573, Y 20.9016, Z -5.5000, A 0.000, B 0.000, C 0.000 }
gfCNCPoint4[6417] = {X 129.7606, Y 20.2049, Z -5.5000, A 0.000, B 0.000, C 0.000 }
gfCNCPoint4[6418] = {X 129.2364, Y 19.3706, Z -5.5000, A 0.000, B 0.000, C 0.000 }
gfCNCPoint4[6419] = {X 128.9110, Y 18.4406, Z -5.5000, A 0.000, B 0.000, C 0.000 }
gfCNCPoint4[6420] = {X 128.8006, Y 17.4615, Z -5.5000, A 0.000, B 0.000, C 0.000 }
gfCNCPoint4[6421] = {X 128.8006, Y 10.4835, Z -5.5000, A 0.000, B 0.000, C 0.000 }
gfCNCPoint4[6422] = {X 128.8808, Y 9.6474, Z -5.5000, A 0.000, B 0.000, C 0.000 }
gfCNCPoint4[6423] = {X 129.1184, Y 8.8418, Z -5.5000, A 0.000, B 0.000, C 0.000 }
gfCNCPoint4[6424] = {X 129.5047, Y 8.0960, Z -5.5000, A 0.000, B 0.000, C 0.000 }
gfCNCPoint4[6425] = {X 130.0257, Y 7.4373, Z -5.5000, A 0.000, B 0.000, C 0.000 }
gfCNCPoint4[6426] = {X 129.6793, Y 7.1049, Z -5.5000, A 0.000, B 0.000, C 0.000 }
gfCNCPoint4[6427] = {X 102.4337, Y 7.1049, Z -5.5000, A 0.000, B 0.000, C 0.000 }
gfCNCPoint4[6428] = {X 102.4337, Y 11.9049, Z -5.5000, A 0.000, B 0.000, C 0.000 }
gfCNCPoint4[6429] = {X 101.3242, Y 11.9049, Z -5.5000, A 0.000, B 0.000, C 0.000 }
gfCNCPoint4[6430] = {X 101.3283, Y 12.0458, Z -5.5000, A 0.000, B 0.000, C 0.000 }
gfCNCPoint4[6431] = {X 101.3297, Y 12.1868, Z -5.5000, A 0.000, B 0.000, C 0.000 }
gfCNCPoint4[6432] = {X 101.3293, Y 13.0462, Z -5.5000, A 0.000, B 0.000, C 0.000 }
gfCNCPoint4[6433] = {X 101.2275, Y 14.1934, Z -5.5000, A 0.000, B 0.000, C 0.000 }
gfCNCPoint4[6434] = {X 100.9460, Y 15.3102, Z -5.5000, A 0.000, B 0.000, C 0.000 }
gfCNCPoint4[6435] = {X 101.0400, Y 15.5443, Z -5.5000, A 0.000, B 0.000, C 0.000 }
gfCNCPoint4[6436] = {X 101.8684, Y 17.5978, Z -5.5000, A 0.000, B 0.000, C 0.000 }
gfCNCPoint4[6437] = {X 102.8000, Y 15.2746, Z -5.5000, A 0.000, B 0.000, C 0.000 }
gfCNCPoint4[6438] = {X 102.5264, Y 14.1691, Z -5.5000, A 0.000, B 0.000, C 0.000 }
gfCNCPoint4[6439] = {X 102.4285, Y 13.0344, Z -5.5000, A 0.000, B 0.000, C 0.000 }
gfCNCPoint4[6440] = {X 102.4283, Y 12.1868, Z -5.5000, A 0.000, B 0.000, C 0.000 }
gfCNCPoint4[6441] = {X 102.4296, Y 12.0458, Z -5.5000, A 0.000, B 0.000, C 0.000 }
gfCNCPoint4[6442] = {X 102.4337, Y 11.9049, Z -5.5000, A 0.000, B 0.000, C 0.000 }
gfCNCPoint4[6443] = {X 102.4337, Y 9.5049, Z -5.5000, A 0.000, B 0.000, C 0.000 }
gfCNCPoint4[6444] = {X 98.1267, Y 9.5049, Z -5.5000, A 0.000, B 0.000, C 0.000 }
gfCNCPoint4[6445] = {X 98.5429, Y 10.2828, Z -5.5000, A 0.000, B 0.000, C 0.000 }
gfCNCPoint4[6446] = {X 98.8123, Y 11.1230, Z -5.5000, A 0.000, B 0.000, C 0.000 }
gfCNCPoint4[6447] = {X 98.9260, Y 11.9979, Z -5.5000, A 0.000, B 0.000, C 0.000 }
gfCNCPoint4[6448] = {X 98.9288, Y 12.0923, Z -5.5000, A 0.000, B 0.000, C 0.000 }
gfCNCPoint4[6449] = {X 98.9297, Y 12.1868, Z -5.5000, A 0.000, B 0.000, C 0.000 }
gfCNCPoint4[6450] = {X 98.9294, Y 13.0237, Z -5.5000, A 0.000, B 0.000, C 0.000 }
gfCNCPoint4[6451] = {X 98.8590, Y 13.8056, Z -5.5000, A 0.000, B 0.000, C 0.000 }
gfCNCPoint4[6452] = {X 98.6640, Y 14.5661, Z -5.5000, A 0.000, B 0.000, C 0.000 }
gfCNCPoint4[6453] = {X 98.3497, Y 15.2855, Z -5.5000, A 0.000, B 0.000, C 0.000 }
gfCNCPoint4[6454] = {X 98.8136, Y 16.4405, Z -5.5000, A 0.000, B 0.000, C 0.000 }
gfCNCPoint4[6455] = {X 101.8739, Y 24.0264, Z -5.5000, A 0.000, B 0.000, C 0.000 }
gfCNCPoint4[6456] = {X 102.9749, Y 21.2869, Z -5.5000, A 0.000, B 0.000, C 0.000 }
gfCNCPoint4[6457] = {X 105.3929, Y 15.2567, Z -5.5000, A 0.000, B 0.000, C 0.000 }
gfCNCPoint4[6458] = {X 105.0868, Y 14.5453, Z -5.5000, A 0.000, B 0.000, C 0.000 }
gfCNCPoint4[6459] = {X 104.8971, Y 13.7945, Z -5.5000, A 0.000, B 0.000, C 0.000 }
gfCNCPoint4[6460] = {X 104.8285, Y 13.0231, Z -5.5000, A 0.000, B 0.000, C 0.000 }
gfCNCPoint4[6461] = {X 104.8283, Y 12.1868, Z -5.5000, A 0.000, B 0.000, C 0.000 }
gfCNCPoint4[6462] = {X 104.8292, Y 12.0923, Z -5.5000, A 0.000, B 0.000, C 0.000 }
gfCNCPoint4[6463] = {X 104.8319, Y 11.9979, Z -5.5000, A 0.000, B 0.000, C 0.000 }
gfCNCPoint4[6464] = {X 104.9456, Y 11.1230, Z -5.5000, A 0.000, B 0.000, C 0.000 }
gfCNCPoint4[6465] = {X 105.2150, Y 10.2828, Z -5.5000, A 0.000, B 0.000, C 0.000 }
gfCNCPoint4[6466] = {X 105.6313, Y 9.5049, Z -5.5000, A 0.000, B 0.000, C 0.000 }
gfCNCPoint4[6467] = {X 102.4337, Y 9.5049, Z -5.5000, A 0.000, B 0.000, C 0.000 }
gfCNCPoint4[6468] = {X 102.4337, Y 7.1049, Z -5.5000, A 0.000, B 0.000, C 0.000 }
gfCNCPoint4[6469] = {X 64.8349, Y 7.1049, Z -5.5000, A 0.000, B 0.000, C 0.000 }
gfCNCPoint4[6470] = {X 65.5946, Y 8.0241, Z -5.5000, A 0.000, B 0.000, C 0.000 }
gfCNCPoint4[6471] = {X 66.1940, Y 9.0550, Z -5.5000, A 0.000, B 0.000, C 0.000 }
gfCNCPoint4[6472] = {X 66.6171, Y 10.1699, Z -5.5000, A 0.000, B 0.000, C 0.000 }
gfCNCPoint4[6473] = {X 66.8305, Y 11.1683, Z -5.5000, A 0.000, B 0.000, C 0.000 }
gfCNCPoint4[6474] = {X 66.9021, Y 12.1868, Z -5.5000, A 0.000, B 0.000, C 0.000 }
gfCNCPoint4[6475] = {X 66.9018, Y 13.0462, Z -5.5000, A 0.000, B 0.000, C 0.000 }
gfCNCPoint4[6476] = {X 66.7773, Y 14.3206, Z -5.5000, A 0.000, B 0.000, C 0.000 }
gfCNCPoint4[6477] = {X 66.4313, Y 15.5535, Z -5.5000, A 0.000, B 0.000, C 0.000 }
gfCNCPoint4[6478] = {X 74.9121, Y 38.2398, Z -5.5000, A 0.000, B 0.000, C 0.000 }
gfCNCPoint4[6479] = {X 75.8042, Y 38.9746, Z -5.5000, A 0.000, B 0.000, C 0.000 }
gfCNCPoint4[6480] = {X 76.5688, Y 39.8413, Z -5.5000, A 0.000, B 0.000, C 0.000 }
gfCNCPoint4[6481] = {X 77.1866, Y 40.8181, Z -5.5000, A 0.000, B 0.000, C 0.000 }
gfCNCPoint4[6482] = {X 77.6421, Y 41.8804, Z -5.5000, A 0.000, B 0.000, C 0.000 }
gfCNCPoint4[6483] = {X 77.9236, Y 43.0013, Z -5.5000, A 0.000, B 0.000, C 0.000 }
gfCNCPoint4[6484] = {X 78.0243, Y 44.1527, Z -5.5000, A 0.000, B 0.000, C 0.000 }
gfCNCPoint4[6485] = {X 78.0245, Y 45.0000, Z -5.5000, A 0.000, B 0.000, C 0.000 }
gfCNCPoint4[6486] = {X 77.9139, Y 46.2642, Z -5.5000, A 0.000, B 0.000, C 0.000 }
gfCNCPoint4[6487] = {X 77.5854, Y 47.4899, Z -5.5000, A 0.000, B 0.000, C 0.000 }
gfCNCPoint4[6488] = {X 77.0491, Y 48.6400, Z -5.5000, A 0.000, B 0.000, C 0.000 }
gfCNCPoint4[6489] = {X 76.3213, Y 49.6795, Z -5.5000, A 0.000, B 0.000, C 0.000 }
gfCNCPoint4[6490] = {X 75.4240, Y 50.5768, Z -5.5000, A 0.000, B 0.000, C 0.000 }
gfCNCPoint4[6491] = {X 74.3845, Y 51.3047, Z -5.5000, A 0.000, B 0.000, C 0.000 }
gfCNCPoint4[6492] = {X 73.2344, Y 51.8410, Z -5.5000, A 0.000, B 0.000, C 0.000 }
gfCNCPoint4[6493] = {X 72.0086, Y 52.1694, Z -5.5000, A 0.000, B 0.000, C 0.000 }
gfCNCPoint4[6494] = {X 70.7445, Y 52.2800, Z -5.5000, A 0.000, B 0.000, C 0.000 }
gfCNCPoint4[6495] = {X 64.1851, Y 52.2800, Z -5.5000, A 0.000, B 0.000, C 0.000 }
gfCNCPoint4[6496] = {X 62.9397, Y 52.1727, Z -5.5000, A 0.000, B 0.000, C 0.000 }
gfCNCPoint4[6497] = {X 61.7311, Y 51.8539, Z -5.5000, A 0.000, B 0.000, C 0.000 }
gfCNCPoint4[6498] = {X 60.5947, Y 51.3330, Z -5.5000, A 0.000, B 0.000, C 0.000 }
gfCNCPoint4[6499] = {X 59.5643, Y 50.6255, Z -5.5000, A 0.000, B 0.000, C 0.000 }
gfCNCPoint4[6500] = {X 58.6700, Y 49.7521, Z -5.5000, A 0.000, B 0.000, C 0.000 }
gfCNCPoint4[6501] = {X 57.9384, Y 48.7385, Z -5.5000, A 0.000, B 0.000, C 0.000 }
gfCNCPoint4[6502] = {X 57.3706, Y 47.5614, Z -5.5000, A 0.000, B 0.000, C 0.000 }
gfCNCPoint4[6503] = {X 57.0224, Y 46.3017, Z -5.5000, A 0.000, B 0.000, C 0.000 }
gfCNCPoint4[6504] = {X 56.9051, Y 45.0000, Z -5.5000, A 0.000, B 0.000, C 0.000 }
gfCNCPoint4[6505] = {X 56.9051, Y 44.2048, Z -5.5000, A 0.000, B 0.000, C 0.000 }
gfCNCPoint4[6506] = {X 56.9286, Y 43.6252, Z -5.5000, A 0.000, B 0.000, C 0.000 }
gfCNCPoint4[6507] = {X 56.9981, Y 43.0492, Z -5.5000, A 0.000, B 0.000, C 0.000 }
gfCNCPoint4[6508] = {X 54.7600, Y 43.0492, Z -5.5000, A 0.000, B 0.000, C 0.000 }
gfCNCPoint4[6509] = {X 54.8275, Y 43.6012, Z -5.5000, A 0.000, B 0.000, C 0.000 }
gfCNCPoint4[6510] = {X 54.8528, Y 44.1567, Z -5.5000, A 0.000, B 0.000, C 0.000 }
gfCNCPoint4[6511] = {X 54.8529, Y 45.0000, Z -5.5000, A 0.000, B 0.000, C 0.000 }
gfCNCPoint4[6512] = {X 54.7356, Y 46.3017, Z -5.5000, A 0.000, B 0.000, C 0.000 }
gfCNCPoint4[6513] = {X 54.3875, Y 47.5614, Z -5.5000, A 0.000, B 0.000, C 0.000 }
gfCNCPoint4[6514] = {X 53.8197, Y 48.7385, Z -5.5000, A 0.000, B 0.000, C 0.000 }
gfCNCPoint4[6515] = {X 53.0880, Y 49.7521, Z -5.5000, A 0.000, B 0.000, C 0.000 }
gfCNCPoint4[6516] = {X 52.1938, Y 50.6255, Z -5.5000, A 0.000, B 0.000, C 0.000 }
gfCNCPoint4[6517] = {X 51.1633, Y 51.3330, Z -5.5000, A 0.000, B 0.000, C 0.000 }
gfCNCPoint4[6518] = {X 50.0270, Y 51.8539, Z -5.5000, A 0.000, B 0.000, C 0.000 }
gfCNCPoint4[6519] = {X 48.8183, Y 52.1727, Z -5.5000, A 0.000, B 0.000, C 0.000 }
gfCNCPoint4[6520] = {X 47.5729, Y 52.2800, Z -5.5000, A 0.000, B 0.000, C 0.000 }
gfCNCPoint4[6521] = {X 40.6393, Y 52.2800, Z -5.5000, A 0.000, B 0.000, C 0.000 }
gfCNCPoint4[6522] = {X 39.4476, Y 52.1818, Z -5.5000, A 0.000, B 0.000, C 0.000 }
gfCNCPoint4[6523] = {X 38.2881, Y 51.8899, Z -5.5000, A 0.000, B 0.000, C 0.000 }
gfCNCPoint4[6524] = {X 37.1919, Y 51.4120, Z -5.5000, A 0.000, B 0.000, C 0.000 }
gfCNCPoint4[6525] = {X 36.1888, Y 50.7612, Z -5.5000, A 0.000, B 0.000, C 0.000 }
gfCNCPoint4[6526] = {X 35.3058, Y 49.9550, Z -5.5000, A 0.000, B 0.000, C 0.000 }
gfCNCPoint4[6527] = {X 34.8234, Y 50.4196, Z -5.5000, A 0.000, B 0.000, C 0.000 }
gfCNCPoint4[6528] = {X 34.3150, Y 50.8555, Z -5.5000, A 0.000, B 0.000, C 0.000 }
gfCNCPoint4[6529] = {X 33.7774, Y 51.2902, Z -5.5000, A 0.000, B 0.000, C 0.000 }
gfCNCPoint4[6530] = {X 32.5188, Y 52.1761, Z -5.5000, A 0.000, B 0.000, C 0.000 }
gfCNCPoint4[6531] = {X 31.1541, Y 52.8878, Z -5.5000, A 0.000, B 0.000, C 0.000 }
gfCNCPoint4[6532] = {X 29.7072, Y 53.4128, Z -5.5000, A 0.000, B 0.000, C 0.000 }
gfCNCPoint4[6533] = {X 28.2036, Y 53.7419, Z -5.5000, A 0.000, B 0.000, C 0.000 }
gfCNCPoint4[6534] = {X 26.6698, Y 53.8692, Z -5.5000, A 0.000, B 0.000, C 0.000 }
gfCNCPoint4[6535] = {X 24.3206, Y 54.9126, Z -5.5000, A 0.000, B 0.000, C 0.000 }
gfCNCPoint4[6536] = {X 21.9038, Y 55.7879, Z -5.5000, A 0.000, B 0.000, C 0.000 }
gfCNCPoint4[6537] = {X 19.5301, Y 56.4637, Z -5.5000, A 0.000, B 0.000, C 0.000 }
gfCNCPoint4[6538] = {X 17.1089, Y 56.9423, Z -5.5000, A 0.000, B 0.000, C 0.000 }
gfCNCPoint4[6539] = {X 14.6566, Y 57.2206, Z -5.5000, A 0.000, B 0.000, C 0.000 }
gfCNCPoint4[6540] = {X 12.1897, Y 57.2967, Z -5.5000, A 0.000, B 0.000, C 0.000 }
gfCNCPoint4[6541] = {X 9.7249, Y 57.1700, Z -5.5000, A 0.000, B 0.000, C 0.000 }
gfCNCPoint4[6542] = {X 8.4102, Y 57.0189, Z -5.5000, A 0.000, B 0.000, C 0.000 }
gfCNCPoint4[6543] = {X 7.1034, Y 56.8100, Z -5.5000, A 0.000, B 0.000, C 0.000 }
gfCNCPoint4[6544] = {X 7.1034, Y 92.8951, Z -5.5000, A 0.000, B 0.000, C 0.000 }
gfCNCPoint4[6545] = {X 116.2647, Y 92.8951, Z -5.5000, A 0.000, B 0.000, C 0.000 }
gfCNCPoint4[6546] = {X 116.9735, Y 91.6539, Z -5.5000, A 0.000, B 0.000, C 0.000 }
gfCNCPoint4[6547] = {X 117.8574, Y 90.5307, Z -5.5000, A 0.000, B 0.000, C 0.000 }
gfCNCPoint4[6548] = {X 118.8970, Y 89.5498, Z -5.5000, A 0.000, B 0.000, C 0.000 }
gfCNCPoint4[6549] = {X 120.0698, Y 88.7328, Z -5.5000, A 0.000, B 0.000, C 0.000 }
gfCNCPoint4[6550] = {X 121.3501, Y 88.0973, Z -5.5000, A 0.000, B 0.000, C 0.000 }
gfCNCPoint4[6551] = {X 122.7100, Y 87.6573, Z -5.5000, A 0.000, B 0.000, C 0.000 }
gfCNCPoint4[6552] = {X 124.1198, Y 87.4223, Z -5.5000, A 0.000, B 0.000, C 0.000 }
gfCNCPoint4[6553] = {X 124.5372, Y 87.3604, Z -5.5000, A 0.000, B 0.000, C 0.000 }
gfCNCPoint4[6554] = {X 125.0280, Y 86.8585, Z -5.5000, A 0.000, B 0.000, C 0.000 }
gfCNCPoint4[6555] = {X 125.5047, Y 86.3433, Z -5.5000, A 0.000, B 0.000, C 0.000 }
gfCNCPoint4[6556] = {X 149.6585, Y 59.8190, Z -5.5000, A 0.000, B 0.000, C 0.000 }
gfCNCPoint4[6557] = {X 149.6295, Y 59.4064, Z -5.5000, A 0.000, B 0.000, C 0.000 }
gfCNCPoint4[6558] = {X 149.6181, Y 58.9930, Z -5.5000, A 0.000, B 0.000, C 0.000 }
gfCNCPoint4[6559] = {X 149.6180, Y 58.0000, Z -5.5000, A 0.000, B 0.000, C 0.000 }
gfCNCPoint4[6560] = {X 149.6915, Y 56.8093, Z -5.5000, A 0.000, B 0.000, C 0.000 }
gfCNCPoint4[6561] = {X 149.9109, Y 55.6367, Z -5.5000, A 0.000, B 0.000, C 0.000 }
gfCNCPoint4[6562] = {X 150.2729, Y 54.5000, Z -5.5000, A 0.000, B 0.000, C 0.000 }
gfCNCPoint4[6563] = {X 150.7719, Y 53.4164, Z -5.5000, A 0.000, B 0.000, C 0.000 }
gfCNCPoint4[6564] = {X 151.5117, Y 52.2488, Z -5.5000, A 0.000, B 0.000, C 0.000 }
gfCNCPoint4[6565] = {X 152.4103, Y 51.1984, Z -5.5000, A 0.000, B 0.000, C 0.000 }
gfCNCPoint4[6566] = {X 153.4493, Y 50.2867, Z -5.5000, A 0.000, B 0.000, C 0.000 }
gfCNCPoint4[6567] = {X 154.6075, Y 49.5323, Z -5.5000, A 0.000, B 0.000, C 0.000 }
gfCNCPoint4[6568] = {X 155.8614, Y 48.9505, Z -5.5000, A 0.000, B 0.000, C 0.000 }
gfCNCPoint4[6569] = {X 157.1854, Y 48.5533, Z -5.5000, A 0.000, B 0.000, C 0.000 }
gfCNCPoint4[6570] = {X 158.2353, Y 48.3785, Z -5.5000, A 0.000, B 0.000, C 0.000 }
gfCNCPoint4[6571] = {X 159.2980, Y 48.3200, Z -5.5000, A 0.000, B 0.000, C 0.000 }
gfCNCPoint4[6572] = {X 176.3026, Y 48.3200, Z -5.5000, A 0.000, B 0.000, C 0.000 }
gfCNCPoint4[6573] = {X 174.9306, Y 47.4865, Z -5.5000, A 0.000, B 0.000, C 0.000 }
gfCNCPoint4[6574] = {X 173.6426, Y 46.5285, Z -5.5000, A 0.000, B 0.000, C 0.000 }
gfCNCPoint4[6575] = {X 172.5427, Y 45.5342, Z -5.5000, A 0.000, B 0.000, C 0.000 }
gfCNCPoint4[6576] = {X 171.5578, Y 44.4259, Z -5.5000, A 0.000, B 0.000, C 0.000 }
gfCNCPoint4[6577] = {X 170.5963, Y 43.0508, Z -5.5000, A 0.000, B 0.000, C 0.000 }
gfCNCPoint4[6578] = {X 169.8116, Y 41.5676, Z -5.5000, A 0.000, B 0.000, C 0.000 }
gfCNCPoint4[6579] = {X 169.2158, Y 39.9990, Z -5.5000, A 0.000, B 0.000, C 0.000 }
gfCNCPoint4[6580] = {X 168.8179, Y 38.3690, Z -5.5000, A 0.000, B 0.000, C 0.000 }
gfCNCPoint4[6581] = {X 168.7077, Y 37.6766, Z -5.5000, A 0.000, B 0.000, C 0.000 }
gfCNCPoint4[6582] = {X 168.5429, Y 36.0108, Z -5.5000, A 0.000, B 0.000, C 0.000 }
gfCNCPoint4[6583] = {X 168.5601, Y 34.3370, Z -5.5000, A 0.000, B 0.000, C 0.000 }
gfCNCPoint4[6584] = {X 168.7592, Y 32.6750, Z -5.5000, A 0.000, B 0.000, C 0.000 }
gfCNCPoint4[6585] = {X 169.1378, Y 31.0444, Z -5.5000, A 0.000, B 0.000, C 0.000 }
gfCNCPoint4[6586] = {X 169.6914, Y 29.4647, Z -5.5000, A 0.000, B 0.000, C 0.000 }
gfCNCPoint4[6587] = {X 170.2633, Y 28.2678, Z -5.5000, A 0.000, B 0.000, C 0.000 }
gfCNCPoint4[6588] = {X 170.9702, Y 27.1453, Z -5.5000, A 0.000, B 0.000, C 0.000 }
gfCNCPoint4[6589] = {X 171.8025, Y 26.1124, Z -5.5000, A 0.000, B 0.000, C 0.000 }
gfCNCPoint4[6590] = {X 172.7490, Y 25.1831, Z -5.5000, A 0.000, B 0.000, C 0.000 }
gfCNCPoint4[6591] = {X 173.7969, Y 24.3697, Z -5.5000, A 0.000, B 0.000, C 0.000 }
gfCNCPoint4[6592] = {X 173.0269, Y 23.7516, Z -5.5000, A 0.000, B 0.000, C 0.000 }
gfCNCPoint4[6593] = {X 172.3970, Y 22.9910, Z -5.5000, A 0.000, B 0.000, C 0.000 }
gfCNCPoint4[6594] = {X 171.9332, Y 22.1192, Z -5.5000, A 0.000, B 0.000, C 0.000 }
gfCNCPoint4[6595] = {X 169.3220, Y 15.7237, Z -5.5000, A 0.000, B 0.000, C 0.000 }
gfCNCPoint4[6596] = {X 169.1088, Y 15.0753, Z -5.5000, A 0.000, B 0.000, C 0.000 }
gfCNCPoint4[6597] = {X 168.9882, Y 14.4035, Z -5.5000, A 0.000, B 0.000, C 0.000 }
gfCNCPoint4[6598] = {X 168.9599, Y 13.8791, Z -5.5000, A 0.000, B 0.000, C 0.000 }
gfCNCPoint4[6599] = {X 168.9882, Y 13.3548, Z -5.5000, A 0.000, B 0.000, C 0.000 }
gfCNCPoint4[6600] = {X 169.1590, Y 12.4995, Z -5.5000, A 0.000, B 0.000, C 0.000 }
gfCNCPoint4[6601] = {X 169.4794, Y 11.6882, Z -5.5000, A 0.000, B 0.000, C 0.000 }
gfCNCPoint4[6602] = {X 169.9391, Y 10.9470, Z -5.5000, A 0.000, B 0.000, C 0.000 }
gfCNCPoint4[6603] = {X 170.6136, Y 10.2179, Z -5.5000, A 0.000, B 0.000, C 0.000 }
gfCNCPoint4[6604] = {X 171.4217, Y 9.6404, Z -5.5000, A 0.000, B 0.000, C 0.000 }
gfCNCPoint4[6605] = {X 172.0576, Y 9.2779, Z -5.5000, A 0.000, B 0.000, C 0.000 }
gfCNCPoint4[6606] = {X 172.9926, Y 8.8771, Z -5.5000, A 0.000, B 0.000, C 0.000 }
gfCNCPoint4[6607] = {X 173.9905, Y 8.6789, Z -5.5000, A 0.000, B 0.000, C 0.000 }
gfCNCPoint4[6608] = {X 175.0077, Y 8.6919, Z -5.5000, A 0.000, B 0.000, C 0.000 }
gfCNCPoint4[6609] = {X 176.0002, Y 8.9156, Z -5.5000, A 0.000, B 0.000, C 0.000 }
gfCNCPoint4[6610] = {X 176.9240, Y 8.5224, Z -5.5000, A 0.000, B 0.000, C 0.000 }
gfCNCPoint4[6611] = {X 179.1587, Y 7.7004, Z -5.5000, A 0.000, B 0.000, C 0.000 }
gfCNCPoint4[6612] = {X 181.4640, Y 7.1049, Z -5.5000, A 0.000, B 0.000, C 0.000 }
gfCNCPoint4[6613] = {X 168.0206, Y 7.1049, Z -5.5000, A 0.000, B 0.000, C 0.000 }
gfCNCPoint4[6614] = {X 168.0206, Y 4.7049, Z -5.5000, A 0.000, B 0.000, C 0.000 }
gfCNCPoint4[6615] = {X 155.1591, Y 4.7049, Z -5.5000, A 0.000, B 0.000, C 0.000 }
gfCNCPoint4[6616] = {X 155.1591, Y 7.1049, Z -5.5000, A 0.000, B 0.000, C 0.000 }
gfCNCPoint4[6617] = {X 137.3636, Y 7.1049, Z -5.5000, A 0.000, B 0.000, C 0.000 }
gfCNCPoint4[6618] = {X 137.5333, Y 7.2912, Z -5.5000, A 0.000, B 0.000, C 0.000 }
gfCNCPoint4[6619] = {X 137.6932, Y 7.4860, Z -5.5000, A 0.000, B 0.000, C 0.000 }
gfCNCPoint4[6620] = {X 154.8295, Y 7.4860, Z -5.5000, A 0.000, B 0.000, C 0.000 }
gfCNCPoint4[6621] = {X 154.9894, Y 7.2912, Z -5.5000, A 0.000, B 0.000, C 0.000 }
gfCNCPoint4[6622] = {X 155.1591, Y 7.1049, Z -5.5000, A 0.000, B 0.000, C 0.000 }
gfCNCPoint4[6623] = {X 155.1591, Y 4.7049, Z -5.5000, A 0.000, B 0.000, C 0.000 }
gfCNCPoint4[6624] = {X 42.6032, Y 4.7049, Z -5.5000, A 0.000, B 0.000, C 0.000 }
gfCNCPoint4[6625] = {X 42.6032, Y 9.5049, Z -5.5000, A 0.000, B 0.000, C 0.000 }
gfCNCPoint4[6626] = {X 36.0460, Y 9.5049, Z -5.5000, A 0.000, B 0.000, C 0.000 }
gfCNCPoint4[6627] = {X 37.0559, Y 11.3879, Z -5.5000, A 0.000, B 0.000, C 0.000 }
gfCNCPoint4[6628] = {X 37.8841, Y 13.3575, Z -5.5000, A 0.000, B 0.000, C 0.000 }
gfCNCPoint4[6629] = {X 38.5469, Y 15.5385, Z -5.5000, A 0.000, B 0.000, C 0.000 }
gfCNCPoint4[6630] = {X 39.0056, Y 17.7713, Z -5.5000, A 0.000, B 0.000, C 0.000 }
gfCNCPoint4[6631] = {X 39.2563, Y 20.0369, Z -5.5000, A 0.000, B 0.000, C 0.000 }
gfCNCPoint4[6632] = {X 39.2969, Y 22.3160, Z -5.5000, A 0.000, B 0.000, C 0.000 }
gfCNCPoint4[6633] = {X 39.1270, Y 24.5892, Z -5.5000, A 0.000, B 0.000, C 0.000 }
gfCNCPoint4[6634] = {X 42.5394, Y 15.4279, Z -5.5000, A 0.000, B 0.000, C 0.000 }
gfCNCPoint4[6635] = {X 42.3081, Y 14.2497, Z -5.5000, A 0.000, B 0.000, C 0.000 }
gfCNCPoint4[6636] = {X 42.2245, Y 13.0519, Z -5.5000, A 0.000, B 0.000, C 0.000 }
gfCNCPoint4[6637] = {X 42.2242, Y 12.1868, Z -5.5000, A 0.000, B 0.000, C 0.000 }
gfCNCPoint4[6638] = {X 42.3194, Y 10.8326, Z -5.5000, A 0.000, B 0.000, C 0.000 }
gfCNCPoint4[6639] = {X 42.6032, Y 9.5049, Z -5.5000, A 0.000, B 0.000, C 0.000 }
gfCNCPoint4[6640] = {X 42.6032, Y 7.1049, Z -5.5000, A 0.000, B 0.000, C 0.000 }
gfCNCPoint4[6641] = {X 31.2116, Y 7.1049, Z -5.5000, A 0.000, B 0.000, C 0.000 }
gfCNCPoint4[6642] = {X 32.2270, Y 8.2450, Z -5.5000, A 0.000, B 0.000, C 0.000 }
gfCNCPoint4[6643] = {X 33.1538, Y 9.4582, Z -5.5000, A 0.000, B 0.000, C 0.000 }
gfCNCPoint4[6644] = {X 33.9868, Y 10.7377, Z -5.5000, A 0.000, B 0.000, C 0.000 }
gfCNCPoint4[6645] = {X 34.8873, Y 12.4161, Z -5.5000, A 0.000, B 0.000, C 0.000 }
gfCNCPoint4[6646] = {X 35.6264, Y 14.1717, Z -5.5000, A 0.000, B 0.000, C 0.000 }
gfCNCPoint4[6647] = {X 36.2231, Y 16.1386, Z -5.5000, A 0.000, B 0.000, C 0.000 }
gfCNCPoint4[6648] = {X 36.6360, Y 18.1521, Z -5.5000, A 0.000, B 0.000, C 0.000 }
gfCNCPoint4[6649] = {X 36.8616, Y 20.1951, Z -5.5000, A 0.000, B 0.000, C 0.000 }
gfCNCPoint4[6650] = {X 36.8978, Y 22.2502, Z -5.5000, A 0.000, B 0.000, C 0.000 }
gfCNCPoint4[6651] = {X 36.7445, Y 24.2999, Z -5.5000, A 0.000, B 0.000, C 0.000 }
gfCNCPoint4[6652] = {X 36.5511, Y 25.5803, Z -5.5000, A 0.000, B 0.000, C 0.000 }
gfCNCPoint4[6653] = {X 36.2836, Y 26.8474, Z -5.5000, A 0.000, B 0.000, C 0.000 }
gfCNCPoint4[6654] = {X 35.8747, Y 28.3067, Z -5.5000, A 0.000, B 0.000, C 0.000 }
gfCNCPoint4[6655] = {X 35.3506, Y 29.7286, Z -5.5000, A 0.000, B 0.000, C 0.000 }
gfCNCPoint4[6656] = {X 34.7146, Y 31.1042, Z -5.5000, A 0.000, B 0.000, C 0.000 }
gfCNCPoint4[6657] = {X 37.2842, Y 36.4125, Z -5.5000, A 0.000, B 0.000, C 0.000 }
gfCNCPoint4[6658] = {X 41.3760, Y 25.4269, Z -5.5000, A 0.000, B 0.000, C 0.000 }
gfCNCPoint4[6659] = {X 45.0743, Y 15.4981, Z -5.5000, A 0.000, B 0.000, C 0.000 }
gfCNCPoint4[6660] = {X 44.7425, Y 14.2852, Z -5.5000, A 0.000, B 0.000, C 0.000 }
gfCNCPoint4[6661] = {X 44.6244, Y 13.0334, Z -5.5000, A 0.000, B 0.000, C 0.000 }
gfCNCPoint4[6662] = {X 44.6242, Y 12.1868, Z -5.5000, A 0.000, B 0.000, C 0.000 }
gfCNCPoint4[6663] = {X 44.6958, Y 11.1683, Z -5.5000, A 0.000, B 0.000, C 0.000 }
gfCNCPoint4[6664] = {X 44.9092, Y 10.1699, Z -5.5000, A 0.000, B 0.000, C 0.000 }
gfCNCPoint4[6665] = {X 45.3323, Y 9.0550, Z -5.5000, A 0.000, B 0.000, C 0.000 }
gfCNCPoint4[6666] = {X 45.9318, Y 8.0241, Z -5.5000, A 0.000, B 0.000, C 0.000 }
gfCNCPoint4[6667] = {X 46.6915, Y 7.1049, Z -5.5000, A 0.000, B 0.000, C 0.000 }
gfCNCPoint4[6668] = {X 42.6032, Y 7.1049, Z -5.5000, A 0.000, B 0.000, C 0.000 }
gfCNCPoint4[6669] = {X 42.6032, Y 4.7049, Z -5.5000, A 0.000, B 0.000, C 0.000 }
gfCNCPoint4[6670] = {X 23.8360, Y 4.7049, Z -5.5000, A 0.000, B 0.000, C 0.000 }
gfCNCPoint4[6671] = {X 25.7640, Y 5.7849, Z -5.5000, A 0.000, B 0.000, C 0.000 }
gfCNCPoint4[6672] = {X 27.5759, Y 7.0501, Z -5.5000, A 0.000, B 0.000, C 0.000 }
gfCNCPoint4[6673] = {X 28.5592, Y 7.8747, Z -5.5000, A 0.000, B 0.000, C 0.000 }
gfCNCPoint4[6674] = {X 29.4808, Y 8.7676, Z -5.5000, A 0.000, B 0.000, C 0.000 }
gfCNCPoint4[6675] = {X 30.6890, Y 10.1629, Z -5.5000, A 0.000, B 0.000, C 0.000 }
gfCNCPoint4[6676] = {X 31.7470, Y 11.6753, Z -5.5000, A 0.000, B 0.000, C 0.000 }
gfCNCPoint4[6677] = {X 32.6434, Y 13.2887, Z -5.5000, A 0.000, B 0.000, C 0.000 }
gfCNCPoint4[6678] = {X 33.3687, Y 14.9859, Z -5.5000, A 0.000, B 0.000, C 0.000 }
gfCNCPoint4[6679] = {X 33.9190, Y 16.8169, Z -5.5000, A 0.000, B 0.000, C 0.000 }
gfCNCPoint4[6680] = {X 34.2908, Y 18.6924, Z -5.5000, A 0.000, B 0.000, C 0.000 }
gfCNCPoint4[6681] = {X 34.4807, Y 20.5948, Z -5.5000, A 0.000, B 0.000, C 0.000 }
gfCNCPoint4[6682] = {X 34.4869, Y 22.5067, Z -5.5000, A 0.000, B 0.000, C 0.000 }
gfCNCPoint4[6683] = {X 34.3093, Y 24.4104, Z -5.5000, A 0.000, B 0.000, C 0.000 }
gfCNCPoint4[6684] = {X 33.9497, Y 26.2881, Z -5.5000, A 0.000, B 0.000, C 0.000 }
gfCNCPoint4[6685] = {X 33.4659, Y 27.9397, Z -5.5000, A 0.000, B 0.000, C 0.000 }
gfCNCPoint4[6686] = {X 32.8134, Y 29.5322, Z -5.5000, A 0.000, B 0.000, C 0.000 }
gfCNCPoint4[6687] = {X 31.9993, Y 31.0485, Z -5.5000, A 0.000, B 0.000, C 0.000 }
gfCNCPoint4[6688] = {X 32.1286, Y 31.2840, Z -5.5000, A 0.000, B 0.000, C 0.000 }
gfCNCPoint4[6689] = {X 32.2510, Y 31.5232, Z -5.5000, A 0.000, B 0.000, C 0.000 }
gfCNCPoint4[6690] = {X 35.3025, Y 37.8269, Z -5.5000, A 0.000, B 0.000, C 0.000 }
gfCNCPoint4[6691] = {X 35.7263, Y 38.8573, Z -5.5000, A 0.000, B 0.000, C 0.000 }
gfCNCPoint4[6692] = {X 36.0224, Y 39.9313, Z -5.5000, A 0.000, B 0.000, C 0.000 }
gfCNCPoint4[6693] = {X 36.1865, Y 41.0332, Z -5.5000, A 0.000, B 0.000, C 0.000 }
gfCNCPoint4[6694] = {X 36.2163, Y 42.1469, Z -5.5000, A 0.000, B 0.000, C 0.000 }
gfCNCPoint4[6695] = {X 36.6303, Y 41.4263, Z -5.5000, A 0.000, B 0.000, C 0.000 }
gfCNCPoint4[6696] = {X 37.1607, Y 40.7863, Z -5.5000, A 0.000, B 0.000, C 0.000 }
gfCNCPoint4[6697] = {X 37.7919, Y 40.2456, Z -5.5000, A 0.000, B 0.000, C 0.000 }
gfCNCPoint4[6698] = {X 38.5057, Y 39.8199, Z -5.5000, A 0.000, B 0.000, C 0.000 }
gfCNCPoint4[6699] = {X 39.0445, Y 38.5341, Z -5.5000, A 0.000, B 0.000, C 0.000 }
gfCNCPoint4[6700] = {X 39.5403, Y 37.2311, Z -5.5000, A 0.000, B 0.000, C 0.000 }
gfCNCPoint4[6701] = {X 47.6703, Y 15.4045, Z -5.5000, A 0.000, B 0.000, C 0.000 }
gfCNCPoint4[6702] = {X 47.3200, Y 14.6512, Z -5.5000, A 0.000, B 0.000, C 0.000 }
gfCNCPoint4[6703] = {X 47.1026, Y 13.8493, Z -5.5000, A 0.000, B 0.000, C 0.000 }
gfCNCPoint4[6704] = {X 47.0244, Y 13.0222, Z -5.5000, A 0.000, B 0.000, C 0.000 }
gfCNCPoint4[6705] = {X 47.0242, Y 12.1868, Z -5.5000, A 0.000, B 0.000, C 0.000 }
gfCNCPoint4[6706] = {X 47.1150, Y 11.2500, Z -5.5000, A 0.000, B 0.000, C 0.000 }
gfCNCPoint4[6707] = {X 47.3839, Y 10.3480, Z -5.5000, A 0.000, B 0.000, C 0.000 }
gfCNCPoint4[6708] = {X 47.8210, Y 9.5144, Z -5.5000, A 0.000, B 0.000, C 0.000 }
gfCNCPoint4[6709] = {X 48.4100, Y 8.7803, Z -5.5000, A 0.000, B 0.000, C 0.000 }
gfCNCPoint4[6710] = {X 49.1545, Y 8.1553, Z -5.5000, A 0.000, B 0.000, C 0.000 }
gfCNCPoint4[6711] = {X 50.0081, Y 7.6902, Z -5.5000, A 0.000, B 0.000, C 0.000 }
gfCNCPoint4[6712] = {X 50.9370, Y 7.4036, Z -5.5000, A 0.000, B 0.000, C 0.000 }
gfCNCPoint4[6713] = {X 51.9042, Y 7.3068, Z -5.5000, A 0.000, B 0.000, C 0.000 }
gfCNCPoint4[6714] = {X 59.6221, Y 7.3068, Z -5.5000, A 0.000, B 0.000, C 0.000 }
gfCNCPoint4[6715] = {X 60.5894, Y 7.4036, Z -5.5000, A 0.000, B 0.000, C 0.000 }
gfCNCPoint4[6716] = {X 61.5182, Y 7.6902, Z -5.5000, A 0.000, B 0.000, C 0.000 }
gfCNCPoint4[6717] = {X 62.3719, Y 8.1553, Z -5.5000, A 0.000, B 0.000, C 0.000 }
gfCNCPoint4[6718] = {X 63.1164, Y 8.7803, Z -5.5000, A 0.000, B 0.000, C 0.000 }
gfCNCPoint4[6719] = {X 63.7054, Y 9.5144, Z -5.5000, A 0.000, B 0.000, C 0.000 }
gfCNCPoint4[6720] = {X 64.1424, Y 10.3480, Z -5.5000, A 0.000, B 0.000, C 0.000 }
gfCNCPoint4[6721] = {X 64.4114, Y 11.2500, Z -5.5000, A 0.000, B 0.000, C 0.000 }
gfCNCPoint4[6722] = {X 64.5021, Y 12.1868, Z -5.5000, A 0.000, B 0.000, C 0.000 }
gfCNCPoint4[6723] = {X 64.5019, Y 13.0237, Z -5.5000, A 0.000, B 0.000, C 0.000 }
gfCNCPoint4[6724] = {X 64.4204, Y 13.8672, Z -5.5000, A 0.000, B 0.000, C 0.000 }
gfCNCPoint4[6725] = {X 64.1942, Y 14.6840, Z -5.5000, A 0.000, B 0.000, C 0.000 }
gfCNCPoint4[6726] = {X 63.8302, Y 15.4492, Z -5.5000, A 0.000, B 0.000, C 0.000 }
gfCNCPoint4[6727] = {X 72.9549, Y 39.8581, Z -5.5000, A 0.000, B 0.000, C 0.000 }
gfCNCPoint4[6728] = {X 73.8447, Y 40.4401, Z -5.5000, A 0.000, B 0.000, C 0.000 }
gfCNCPoint4[6729] = {X 74.5873, Y 41.2010, Z -5.5000, A 0.000, B 0.000, C 0.000 }
gfCNCPoint4[6730] = {X 75.1475, Y 42.1047, Z -5.5000, A 0.000, B 0.000, C 0.000 }
gfCNCPoint4[6731] = {X 75.4987, Y 43.1082, Z -5.5000, A 0.000, B 0.000, C 0.000 }
gfCNCPoint4[6732] = {X 75.6243, Y 44.1640, Z -5.5000, A 0.000, B 0.000, C 0.000 }
gfCNCPoint4[6733] = {X 75.6245, Y 45.0000, Z -5.5000, A 0.000, B 0.000, C 0.000 }
gfCNCPoint4[6734] = {X 75.5307, Y 45.9520, Z -5.5000, A 0.000, B 0.000, C 0.000 }
gfCNCPoint4[6735] = {X 75.2530, Y 46.8675, Z -5.5000, A 0.000, B 0.000, C 0.000 }
gfCNCPoint4[6736] = {X 74.8020, Y 47.7112, Z -5.5000, A 0.000, B 0.000, C 0.000 }
gfCNCPoint4[6737] = {X 74.1951, Y 48.4507, Z -5.5000, A 0.000, B 0.000, C 0.000 }
gfCNCPoint4[6738] = {X 73.4556, Y 49.0576, Z -5.5000, A 0.000, B 0.000, C 0.000 }
gfCNCPoint4[6739] = {X 72.6120, Y 49.5085, Z -5.5000, A 0.000, B 0.000, C 0.000 }
gfCNCPoint4[6740] = {X 71.6965, Y 49.7862, Z -5.5000, A 0.000, B 0.000, C 0.000 }
gfCNCPoint4[6741] = {X 70.7445, Y 49.8800, Z -5.5000, A 0.000, B 0.000, C 0.000 }
gfCNCPoint4[6742] = {X 64.1851, Y 49.8800, Z -5.5000, A 0.000, B 0.000, C 0.000 }
gfCNCPoint4[6743] = {X 63.2331, Y 49.7862, Z -5.5000, A 0.000, B 0.000, C 0.000 }
gfCNCPoint4[6744] = {X 62.3176, Y 49.5085, Z -5.5000, A 0.000, B 0.000, C 0.000 }
gfCNCPoint4[6745] = {X 61.4740, Y 49.0576, Z -5.5000, A 0.000, B 0.000, C 0.000 }
gfCNCPoint4[6746] = {X 60.7345, Y 48.4507, Z -5.5000, A 0.000, B 0.000, C 0.000 }
gfCNCPoint4[6747] = {X 60.1276, Y 47.7112, Z -5.5000, A 0.000, B 0.000, C 0.000 }
gfCNCPoint4[6748] = {X 59.6766, Y 46.8675, Z -5.5000, A 0.000, B 0.000, C 0.000 }
gfCNCPoint4[6749] = {X 59.3989, Y 45.9520, Z -5.5000, A 0.000, B 0.000, C 0.000 }
gfCNCPoint4[6750] = {X 59.3051, Y 45.0000, Z -5.5000, A 0.000, B 0.000, C 0.000 }
gfCNCPoint4[6751] = {X 59.3052, Y 44.2028, Z -5.5000, A 0.000, B 0.000, C 0.000 }
gfCNCPoint4[6752] = {X 59.3847, Y 43.3312, Z -5.5000, A 0.000, B 0.000, C 0.000 }
gfCNCPoint4[6753] = {X 59.6187, Y 42.4878, Z -5.5000, A 0.000, B 0.000, C 0.000 }
gfCNCPoint4[6754] = {X 59.9996, Y 41.6997, Z -5.5000, A 0.000, B 0.000, C 0.000 }
gfCNCPoint4[6755] = {X 59.6153, Y 40.6492, Z -5.5000, A 0.000, B 0.000, C 0.000 }
gfCNCPoint4[6756] = {X 52.4667, Y 40.6492, Z -5.5000, A 0.000, B 0.000, C 0.000 }
gfCNCPoint4[6757] = {X 51.9471, Y 42.0452, Z -5.5000, A 0.000, B 0.000, C 0.000 }
gfCNCPoint4[6758] = {X 52.2217, Y 42.7245, Z -5.5000, A 0.000, B 0.000, C 0.000 }
gfCNCPoint4[6759] = {X 52.3915, Y 43.4371, Z -5.5000, A 0.000, B 0.000, C 0.000 }
gfCNCPoint4[6760] = {X 52.4528, Y 44.1672, Z -5.5000, A 0.000, B 0.000, C 0.000 }
gfCNCPoint4[6761] = {X 52.4529, Y 45.0000, Z -5.5000, A 0.000, B 0.000, C 0.000 }
gfCNCPoint4[6762] = {X 52.3592, Y 45.9520, Z -5.5000, A 0.000, B 0.000, C 0.000 }
gfCNCPoint4[6763] = {X 52.0815, Y 46.8675, Z -5.5000, A 0.000, B 0.000, C 0.000 }
gfCNCPoint4[6764] = {X 51.6305, Y 47.7112, Z -5.5000, A 0.000, B 0.000, C 0.000 }
gfCNCPoint4[6765] = {X 51.0236, Y 48.4507, Z -5.5000, A 0.000, B 0.000, C 0.000 }
gfCNCPoint4[6766] = {X 50.2841, Y 49.0576, Z -5.5000, A 0.000, B 0.000, C 0.000 }
gfCNCPoint4[6767] = {X 49.4404, Y 49.5085, Z -5.5000, A 0.000, B 0.000, C 0.000 }
gfCNCPoint4[6768] = {X 48.5250, Y 49.7862, Z -5.5000, A 0.000, B 0.000, C 0.000 }
gfCNCPoint4[6769] = {X 47.5729, Y 49.8800, Z -5.5000, A 0.000, B 0.000, C 0.000 }
gfCNCPoint4[6770] = {X 40.6393, Y 49.8800, Z -5.5000, A 0.000, B 0.000, C 0.000 }
gfCNCPoint4[6771] = {X 39.6433, Y 49.7773, Z -5.5000, A 0.000, B 0.000, C 0.000 }
gfCNCPoint4[6772] = {X 38.6892, Y 49.4734, Z -5.5000, A 0.000, B 0.000, C 0.000 }
gfCNCPoint4[6773] = {X 37.8173, Y 48.9813, Z -5.5000, A 0.000, B 0.000, C 0.000 }
gfCNCPoint4[6774] = {X 37.0641, Y 48.3215, Z -5.5000, A 0.000, B 0.000, C 0.000 }
gfCNCPoint4[6775] = {X 36.5085, Y 47.5983, Z -5.5000, A 0.000, B 0.000, C 0.000 }
gfCNCPoint4[6776] = {X 36.0972, Y 46.7843, Z -5.5000, A 0.000, B 0.000, C 0.000 }
gfCNCPoint4[6777] = {X 35.8445, Y 45.9080, Z -5.5000, A 0.000, B 0.000, C 0.000 }
gfCNCPoint4[6778] = {X 35.7593, Y 45.0000, Z -5.5000, A 0.000, B 0.000, C 0.000 }
gfCNCPoint4[6779] = {X 35.7593, Y 44.7148, Z -5.5000, A 0.000, B 0.000, C 0.000 }
gfCNCPoint4[6780] = {X 36.2393, Y 44.7148, Z -5.5000, A 0.000, B 0.000, C 0.000 }
gfCNCPoint4[6781] = {X 36.2397, Y 44.1483, Z -5.5000, A 0.000, B 0.000, C 0.000 }
gfCNCPoint4[6782] = {X 36.3680, Y 43.1523, Z -5.5000, A 0.000, B 0.000, C 0.000 }
gfCNCPoint4[6783] = {X 36.7188, Y 42.2113, Z -5.5000, A 0.000, B 0.000, C 0.000 }
gfCNCPoint4[6784] = {X 37.2738, Y 41.3744, Z -5.5000, A 0.000, B 0.000, C 0.000 }
gfCNCPoint4[6785] = {X 38.0041, Y 40.6852, Z -5.5000, A 0.000, B 0.000, C 0.000 }
gfCNCPoint4[6786] = {X 38.8717, Y 40.1794, Z -5.5000, A 0.000, B 0.000, C 0.000 }
gfCNCPoint4[6787] = {X 39.4555, Y 38.7989, Z -5.5000, A 0.000, B 0.000, C 0.000 }
gfCNCPoint4[6788] = {X 39.9901, Y 37.3987, Z -5.5000, A 0.000, B 0.000, C 0.000 }
gfCNCPoint4[6789] = {X 48.2011, Y 15.3544, Z -5.5000, A 0.000, B 0.000, C 0.000 }
gfCNCPoint4[6790] = {X 47.8187, Y 14.6115, Z -5.5000, A 0.000, B 0.000, C 0.000 }
gfCNCPoint4[6791] = {X 47.5835, Y 13.8097, Z -5.5000, A 0.000, B 0.000, C 0.000 }
gfCNCPoint4[6792] = {X 47.5042, Y 12.9779, Z -5.5000, A 0.000, B 0.000, C 0.000 }
gfCNCPoint4[6793] = {X 47.5042, Y 12.1868, Z -5.5000, A 0.000, B 0.000, C 0.000 }
gfCNCPoint4[6794] = {X 47.6145, Y 11.2077, Z -5.5000, A 0.000, B 0.000, C 0.000 }
gfCNCPoint4[6795] = {X 47.9400, Y 10.2777, Z -5.5000, A 0.000, B 0.000, C 0.000 }
gfCNCPoint4[6796] = {X 48.4642, Y 9.4435, Z -5.5000, A 0.000, B 0.000, C 0.000 }
gfCNCPoint4[6797] = {X 49.1609, Y 8.7468, Z -5.5000, A 0.000, B 0.000, C 0.000 }
gfCNCPoint4[6798] = {X 49.9951, Y 8.2226, Z -5.5000, A 0.000, B 0.000, C 0.000 }
gfCNCPoint4[6799] = {X 50.9251, Y 7.8971, Z -5.5000, A 0.000, B 0.000, C 0.000 }
gfCNCPoint4[6800] = {X 51.9042, Y 7.7868, Z -5.5000, A 0.000, B 0.000, C 0.000 }
gfCNCPoint4[6801] = {X 59.6221, Y 7.7868, Z -5.5000, A 0.000, B 0.000, C 0.000 }
gfCNCPoint4[6802] = {X 60.6012, Y 7.8971, Z -5.5000, A 0.000, B 0.000, C 0.000 }
gfCNCPoint4[6803] = {X 61.5312, Y 8.2226, Z -5.5000, A 0.000, B 0.000, C 0.000 }
gfCNCPoint4[6804] = {X 62.3655, Y 8.7468, Z -5.5000, A 0.000, B 0.000, C 0.000 }
gfCNCPoint4[6805] = {X 63.0622, Y 9.4435, Z -5.5000, A 0.000, B 0.000, C 0.000 }
gfCNCPoint4[6806] = {X 63.5864, Y 10.2777, Z -5.5000, A 0.000, B 0.000, C 0.000 }
gfCNCPoint4[6807] = {X 63.9118, Y 11.2077, Z -5.5000, A 0.000, B 0.000, C 0.000 }
gfCNCPoint4[6808] = {X 64.0221, Y 12.1868, Z -5.5000, A 0.000, B 0.000, C 0.000 }
gfCNCPoint4[6809] = {X 64.0219, Y 13.0233, Z -5.5000, A 0.000, B 0.000, C 0.000 }
gfCNCPoint4[6810] = {X 63.9336, Y 13.8562, Z -5.5000, A 0.000, B 0.000, C 0.000 }
gfCNCPoint4[6811] = {X 63.6891, Y 14.6572, Z -5.5000, A 0.000, B 0.000, C 0.000 }
gfCNCPoint4[6812] = {X 63.2972, Y 15.3974, Z -5.5000, A 0.000, B 0.000, C 0.000 }
gfCNCPoint4[6813] = {X 63.5011, Y 15.9354, Z -5.5000, A 0.000, B 0.000, C 0.000 }
gfCNCPoint4[6814] = {X 66.3154, Y 23.4036, Z -5.5000, A 0.000, B 0.000, C 0.000 }
gfCNCPoint4[6815] = {X 72.2847, Y 39.4717, Z -5.5000, A 0.000, B 0.000, C 0.000 }
gfCNCPoint4[6816] = {X 72.5778, Y 40.2089, Z -5.5000, A 0.000, B 0.000, C 0.000 }
gfCNCPoint4[6817] = {X 73.4352, Y 40.7274, Z -5.5000, A 0.000, B 0.000, C 0.000 }
gfCNCPoint4[6818] = {X 74.1530, Y 41.4264, Z -5.5000, A 0.000, B 0.000, C 0.000 }
gfCNCPoint4[6819] = {X 74.6941, Y 42.2697, Z -5.5000, A 0.000, B 0.000, C 0.000 }
gfCNCPoint4[6820] = {X 75.0304, Y 43.2135, Z -5.5000, A 0.000, B 0.000, C 0.000 }
gfCNCPoint4[6821] = {X 75.1445, Y 44.2089, Z -5.5000, A 0.000, B 0.000, C 0.000 }
gfCNCPoint4[6822] = {X 75.1445, Y 45.0000, Z -5.5000, A 0.000, B 0.000, C 0.000 }
gfCNCPoint4[6823] = {X 75.0341, Y 45.9791, Z -5.5000, A 0.000, B 0.000, C 0.000 }
gfCNCPoint4[6824] = {X 74.7087, Y 46.9091, Z -5.5000, A 0.000, B 0.000, C 0.000 }
gfCNCPoint4[6825] = {X 74.1845, Y 47.7434, Z -5.5000, A 0.000, B 0.000, C 0.000 }
gfCNCPoint4[6826] = {X 73.4878, Y 48.4401, Z -5.5000, A 0.000, B 0.000, C 0.000 }
gfCNCPoint4[6827] = {X 72.6535, Y 48.9643, Z -5.5000, A 0.000, B 0.000, C 0.000 }
gfCNCPoint4[6828] = {X 71.7236, Y 49.2897, Z -5.5000, A 0.000, B 0.000, C 0.000 }
gfCNCPoint4[6829] = {X 70.7445, Y 49.4000, Z -5.5000, A 0.000, B 0.000, C 0.000 }
gfCNCPoint4[6830] = {X 64.1851, Y 49.4000, Z -5.5000, A 0.000, B 0.000, C 0.000 }
gfCNCPoint4[6831] = {X 63.2060, Y 49.2897, Z -5.5000, A 0.000, B 0.000, C 0.000 }
gfCNCPoint4[6832] = {X 62.2760, Y 48.9643, Z -5.5000, A 0.000, B 0.000, C 0.000 }
gfCNCPoint4[6833] = {X 61.4418, Y 48.4401, Z -5.5000, A 0.000, B 0.000, C 0.000 }
gfCNCPoint4[6834] = {X 60.7451, Y 47.7434, Z -5.5000, A 0.000, B 0.000, C 0.000 }
gfCNCPoint4[6835] = {X 60.2209, Y 46.9091, Z -5.5000, A 0.000, B 0.000, C 0.000 }
gfCNCPoint4[6836] = {X 59.8955, Y 45.9791, Z -5.5000, A 0.000, B 0.000, C 0.000 }
gfCNCPoint4[6837] = {X 59.7851, Y 45.0000, Z -5.5000, A 0.000, B 0.000, C 0.000 }
gfCNCPoint4[6838] = {X 59.7856, Y 44.1483, Z -5.5000, A 0.000, B 0.000, C 0.000 }
gfCNCPoint4[6839] = {X 59.8783, Y 43.3080, Z -5.5000, A 0.000, B 0.000, C 0.000 }
gfCNCPoint4[6840] = {X 60.1301, Y 42.5009, Z -5.5000, A 0.000, B 0.000, C 0.000 }
gfCNCPoint4[6841] = {X 60.5316, Y 41.7569, Z -5.5000, A 0.000, B 0.000, C 0.000 }
gfCNCPoint4[6842] = {X 59.9509, Y 40.1692, Z -5.5000, A 0.000, B 0.000, C 0.000 }
gfCNCPoint4[6843] = {X 52.1332, Y 40.1692, Z -5.5000, A 0.000, B 0.000, C 0.000 }
gfCNCPoint4[6844] = {X 51.4227, Y 42.0782, Z -5.5000, A 0.000, B 0.000, C 0.000 }
gfCNCPoint4[6845] = {X 51.7255, Y 42.7540, Z -5.5000, A 0.000, B 0.000, C 0.000 }
gfCNCPoint4[6846] = {X 51.9106, Y 43.4710, Z -5.5000, A 0.000, B 0.000, C 0.000 }
gfCNCPoint4[6847] = {X 51.9729, Y 44.2089, Z -5.5000, A 0.000, B 0.000, C 0.000 }
gfCNCPoint4[6848] = {X 51.9729, Y 45.0000, Z -5.5000, A 0.000, B 0.000, C 0.000 }
gfCNCPoint4[6849] = {X 51.8626, Y 45.9791, Z -5.5000, A 0.000, B 0.000, C 0.000 }
gfCNCPoint4[6850] = {X 51.5372, Y 46.9091, Z -5.5000, A 0.000, B 0.000, C 0.000 }
gfCNCPoint4[6851] = {X 51.0130, Y 47.7434, Z -5.5000, A 0.000, B 0.000, C 0.000 }
gfCNCPoint4[6852] = {X 50.3163, Y 48.4401, Z -5.5000, A 0.000, B 0.000, C 0.000 }
gfCNCPoint4[6853] = {X 49.4820, Y 48.9643, Z -5.5000, A 0.000, B 0.000, C 0.000 }
gfCNCPoint4[6854] = {X 48.5520, Y 49.2897, Z -5.5000, A 0.000, B 0.000, C 0.000 }
gfCNCPoint4[6855] = {X 47.5729, Y 49.4000, Z -5.5000, A 0.000, B 0.000, C 0.000 }
gfCNCPoint4[6856] = {X 40.6393, Y 49.4000, Z -5.5000, A 0.000, B 0.000, C 0.000 }
gfCNCPoint4[6857] = {X 39.6602, Y 49.2897, Z -5.5000, A 0.000, B 0.000, C 0.000 }
gfCNCPoint4[6858] = {X 38.7302, Y 48.9643, Z -5.5000, A 0.000, B 0.000, C 0.000 }
gfCNCPoint4[6859] = {X 37.8959, Y 48.4401, Z -5.5000, A 0.000, B 0.000, C 0.000 }
gfCNCPoint4[6860] = {X 37.1992, Y 47.7434, Z -5.5000, A 0.000, B 0.000, C 0.000 }
gfCNCPoint4[6861] = {X 36.6750, Y 46.9091, Z -5.5000, A 0.000, B 0.000, C 0.000 }
gfCNCPoint4[6862] = {X 36.3496, Y 45.9791, Z -5.5000, A 0.000, B 0.000, C 0.000 }
gfCNCPoint4[6863] = {X 36.2393, Y 45.0000, Z -5.5000, A 0.000, B 0.000, C 0.000 }
gfCNCPoint4[6864] = {X 36.2393, Y 44.7148, Z -5.5000, A 0.000, B 0.000, C 0.000 }
gfCNCPoint4[6865] = {X 35.7593, Y 44.7148, Z -5.5000, A 0.000, B 0.000, C 0.000 }
gfCNCPoint4[6866] = {X 35.2211, Y 46.0074, Z -5.5000, A 0.000, B 0.000, C 0.000 }
gfCNCPoint4[6867] = {X 34.4930, Y 47.2034, Z -5.5000, A 0.000, B 0.000, C 0.000 }
gfCNCPoint4[6868] = {X 33.5918, Y 48.2750, Z -5.5000, A 0.000, B 0.000, C 0.000 }
gfCNCPoint4[6869] = {X 33.2092, Y 48.6435, Z -5.5000, A 0.000, B 0.000, C 0.000 }
gfCNCPoint4[6870] = {X 32.8060, Y 48.9892, Z -5.5000, A 0.000, B 0.000, C 0.000 }
gfCNCPoint4[6871] = {X 32.2689, Y 49.4235, Z -5.5000, A 0.000, B 0.000, C 0.000 }
gfCNCPoint4[6872] = {X 31.1825, Y 50.1792, Z -5.5000, A 0.000, B 0.000, C 0.000 }
gfCNCPoint4[6873] = {X 29.9990, Y 50.7715, Z -5.5000, A 0.000, B 0.000, C 0.000 }
gfCNCPoint4[6874] = {X 28.7429, Y 51.1881, Z -5.5000, A 0.000, B 0.000, C 0.000 }
gfCNCPoint4[6875] = {X 27.4400, Y 51.4204, Z -5.5000, A 0.000, B 0.000, C 0.000 }
gfCNCPoint4[6876] = {X 26.1173, Y 51.4637, Z -5.5000, A 0.000, B 0.000, C 0.000 }
gfCNCPoint4[6877] = {X 23.6786, Y 52.5826, Z -5.5000, A 0.000, B 0.000, C 0.000 }
gfCNCPoint4[6878] = {X 21.1594, Y 53.5062, Z -5.5000, A 0.000, B 0.000, C 0.000 }
gfCNCPoint4[6879] = {X 18.9477, Y 54.1353, Z -5.5000, A 0.000, B 0.000, C 0.000 }
gfCNCPoint4[6880] = {X 16.6914, Y 54.5783, Z -5.5000, A 0.000, B 0.000, C 0.000 }
gfCNCPoint4[6881] = {X 14.4060, Y 54.8323, Z -5.5000, A 0.000, B 0.000, C 0.000 }
gfCNCPoint4[6882] = {X 12.1075, Y 54.8955, Z -5.5000, A 0.000, B 0.000, C 0.000 }
gfCNCPoint4[6883] = {X 9.8116, Y 54.7674, Z -5.5000, A 0.000, B 0.000, C 0.000 }
gfCNCPoint4[6884] = {X 7.5343, Y 54.4490, Z -5.5000, A 0.000, B 0.000, C 0.000 }
gfCNCPoint4[6885] = {X 7.1098, Y 54.3681, Z -5.5000, A 0.000, B 0.000, C 0.000 }
gfCNCPoint4[6886] = {X 6.6867, Y 54.2806, Z -5.5000, A 0.000, B 0.000, C 0.000 }
gfCNCPoint4[6887] = {X 5.6889, Y 54.0444, Z -5.5000, A 0.000, B 0.000, C 0.000 }
gfCNCPoint4[6888] = {X 4.7034, Y 53.7611, Z -5.5000, A 0.000, B 0.000, C 0.000 }
gfCNCPoint4[6889] = {X 4.7034, Y 95.2951, Z -5.5000, A 0.000, B 0.000, C 0.000 }
gfCNCPoint4[6890] = {X 117.9387, Y 95.2951, Z -5.5000, A 0.000, B 0.000, C 0.000 }
gfCNCPoint4[6891] = {X 118.3609, Y 94.0791, Z -5.5000, A 0.000, B 0.000, C 0.000 }
gfCNCPoint4[6892] = {X 118.9908, Y 92.9565, Z -5.5000, A 0.000, B 0.000, C 0.000 }
gfCNCPoint4[6893] = {X 119.8085, Y 91.9623, Z -5.5000, A 0.000, B 0.000, C 0.000 }
gfCNCPoint4[6894] = {X 120.7886, Y 91.1277, Z -5.5000, A 0.000, B 0.000, C 0.000 }
gfCNCPoint4[6895] = {X 121.9003, Y 90.4788, Z -5.5000, A 0.000, B 0.000, C 0.000 }
gfCNCPoint4[6896] = {X 123.1089, Y 90.0359, Z -5.5000, A 0.000, B 0.000, C 0.000 }
gfCNCPoint4[6897] = {X 124.3766, Y 89.8127, Z -5.5000, A 0.000, B 0.000, C 0.000 }
gfCNCPoint4[6898] = {X 124.4935, Y 89.7932, Z -5.5000, A 0.000, B 0.000, C 0.000 }
gfCNCPoint4[6899] = {X 125.0314, Y 89.7134, Z -5.5000, A 0.000, B 0.000, C 0.000 }
gfCNCPoint4[6900] = {X 125.3489, Y 89.6665, Z -5.5000, A 0.000, B 0.000, C 0.000 }
gfCNCPoint4[6901] = {X 125.6645, Y 89.6086, Z -5.5000, A 0.000, B 0.000, C 0.000 }
gfCNCPoint4[6902] = {X 126.4913, Y 88.7983, Z -5.5000, A 0.000, B 0.000, C 0.000 }
gfCNCPoint4[6903] = {X 127.2837, Y 87.9542, Z -5.5000, A 0.000, B 0.000, C 0.000 }
gfCNCPoint4[6904] = {X 152.2075, Y 60.5844, Z -5.5000, A 0.000, B 0.000, C 0.000 }
gfCNCPoint4[6905] = {X 152.0684, Y 59.7897, Z -5.5000, A 0.000, B 0.000, C 0.000 }
gfCNCPoint4[6906] = {X 152.0181, Y 58.9845, Z -5.5000, A 0.000, B 0.000, C 0.000 }
gfCNCPoint4[6907] = {X 152.0180, Y 58.0000, Z -5.5000, A 0.000, B 0.000, C 0.000 }
gfCNCPoint4[6908] = {X 152.1286, Y 56.7358, Z -5.5000, A 0.000, B 0.000, C 0.000 }
gfCNCPoint4[6909] = {X 152.4570, Y 55.5101, Z -5.5000, A 0.000, B 0.000, C 0.000 }
gfCNCPoint4[6910] = {X 152.9933, Y 54.3600, Z -5.5000, A 0.000, B 0.000, C 0.000 }
gfCNCPoint4[6911] = {X 153.7212, Y 53.3205, Z -5.5000, A 0.000, B 0.000, C 0.000 }
gfCNCPoint4[6912] = {X 154.6185, Y 52.4232, Z -5.5000, A 0.000, B 0.000, C 0.000 }
gfCNCPoint4[6913] = {X 155.6580, Y 51.6953, Z -5.5000, A 0.000, B 0.000, C 0.000 }
gfCNCPoint4[6914] = {X 156.8081, Y 51.1590, Z -5.5000, A 0.000, B 0.000, C 0.000 }
gfCNCPoint4[6915] = {X 158.0338, Y 50.8306, Z -5.5000, A 0.000, B 0.000, C 0.000 }
gfCNCPoint4[6916] = {X 159.2980, Y 50.7200, Z -5.5000, A 0.000, B 0.000, C 0.000 }
gfCNCPoint4[6917] = {X 178.5335, Y 50.7200, Z -5.5000, A 0.000, B 0.000, C 0.000 }
gfCNCPoint4[6918] = {X 179.7875, Y 50.8288, Z -5.5000, A 0.000, B 0.000, C 0.000 }
gfCNCPoint4[6919] = {X 181.0040, Y 51.1520, Z -5.5000, A 0.000, B 0.000, C 0.000 }
gfCNCPoint4[6920] = {X 182.1467, Y 51.6799, Z -5.5000, A 0.000, B 0.000, C 0.000 }
gfCNCPoint4[6921] = {X 183.1813, Y 52.3968, Z -5.5000, A 0.000, B 0.000, C 0.000 }
gfCNCPoint4[6922] = {X 184.0890, Y 53.2953, Z -5.5000, A 0.000, B 0.000, C 0.000 }
gfCNCPoint4[6923] = {X 184.8258, Y 54.3386, Z -5.5000, A 0.000, B 0.000, C 0.000 }
gfCNCPoint4[6924] = {X 185.3688, Y 55.4946, Z -5.5000, A 0.000, B 0.000, C 0.000 }
gfCNCPoint4[6925] = {X 185.7015, Y 56.7277, Z -5.5000, A 0.000, B 0.000, C 0.000 }
gfCNCPoint4[6926] = {X 185.8135, Y 58.0000, Z -5.5000, A 0.000, B 0.000, C 0.000 }
gfCNCPoint4[6927] = {X 185.8133, Y 58.9942, Z -5.5000, A 0.000, B 0.000, C 0.000 }
gfCNCPoint4[6928] = {X 185.7648, Y 59.7748, Z -5.5000, A 0.000, B 0.000, C 0.000 }
gfCNCPoint4[6929] = {X 185.6329, Y 60.5456, Z -5.5000, A 0.000, B 0.000, C 0.000 }
gfCNCPoint4[6930] = {X 211.6617, Y 88.9546, Z -5.5000, A 0.000, B 0.000, C 0.000 }
gfCNCPoint4[6931] = {X 212.0335, Y 89.3390, Z -5.5000, A 0.000, B 0.000, C 0.000 }
gfCNCPoint4[6932] = {X 212.4255, Y 89.7027, Z -5.5000, A 0.000, B 0.000, C 0.000 }
gfCNCPoint4[6933] = {X 212.6034, Y 89.7408, Z -5.5000, A 0.000, B 0.000, C 0.000 }
gfCNCPoint4[6934] = {X 213.4473, Y 89.8471, Z -5.5000, A 0.000, B 0.000, C 0.000 }
gfCNCPoint4[6935] = {X 214.4299, Y 89.7702, Z -5.5000, A 0.000, B 0.000, C 0.000 }
gfCNCPoint4[6936] = {X 215.4139, Y 89.7165, Z -5.5000, A 0.000, B 0.000, C 0.000 }
gfCNCPoint4[6937] = {X 215.6260, Y 89.6933, Z -5.5000, A 0.000, B 0.000, C 0.000 }
gfCNCPoint4[6938] = {X 215.8210, Y 89.6065, Z -5.5000, A 0.000, B 0.000, C 0.000 }
gfCNCPoint4[6939] = {X 239.3458, Y 74.5357, Z -5.5000, A 0.000, B 0.000, C 0.000 }
gfCNCPoint4[6940] = {X 220.5437, Y 67.1573, Z -5.5000, A 0.000, B 0.000, C 0.000 }
gfCNCPoint4[6941] = {X 219.0950, Y 66.6711, Z -5.5000, A 0.000, B 0.000, C 0.000 }
gfCNCPoint4[6942] = {X 217.6001, Y 66.3538, Z -5.5000, A 0.000, B 0.000, C 0.000 }
gfCNCPoint4[6943] = {X 216.0788, Y 66.2097, Z -5.5000, A 0.000, B 0.000, C 0.000 }
gfCNCPoint4[6944] = {X 214.8521, Y 66.0623, Z -5.5000, A 0.000, B 0.000, C 0.000 }
gfCNCPoint4[6945] = {X 213.6680, Y 65.7096, Z -5.5000, A 0.000, B 0.000, C 0.000 }
gfCNCPoint4[6946] = {X 212.5606, Y 65.1617, Z -5.5000, A 0.000, B 0.000, C 0.000 }
gfCNCPoint4[6947] = {X 211.5618, Y 64.4345, Z -5.5000, A 0.000, B 0.000, C 0.000 }
gfCNCPoint4[6948] = {X 210.7004, Y 63.5489, Z -5.5000, A 0.000, B 0.000, C 0.000 }
gfCNCPoint4[6949] = {X 210.0011, Y 62.5303, Z -5.5000, A 0.000, B 0.000, C 0.000 }
gfCNCPoint4[6950] = {X 209.4841, Y 61.4082, Z -5.5000, A 0.000, B 0.000, C 0.000 }
gfCNCPoint4[6951] = {X 209.1643, Y 60.2148, Z -5.5000, A 0.000, B 0.000, C 0.000 }
gfCNCPoint4[6952] = {X 209.0510, Y 58.9845, Z -5.5000, A 0.000, B 0.000, C 0.000 }
gfCNCPoint4[6953] = {X 209.0508, Y 58.0000, Z -5.5000, A 0.000, B 0.000, C 0.000 }
gfCNCPoint4[6954] = {X 209.1477, Y 56.8162, Z -5.5000, A 0.000, B 0.000, C 0.000 }
gfCNCPoint4[6955] = {X 209.4358, Y 55.6638, Z -5.5000, A 0.000, B 0.000, C 0.000 }
gfCNCPoint4[6956] = {X 209.9075, Y 54.5737, Z -5.5000, A 0.000, B 0.000, C 0.000 }
gfCNCPoint4[6957] = {X 210.5502, Y 53.5748, Z -5.5000, A 0.000, B 0.000, C 0.000 }
gfCNCPoint4[6958] = {X 211.3467, Y 52.6937, Z -5.5000, A 0.000, B 0.000, C 0.000 }
gfCNCPoint4[6959] = {X 212.2759, Y 51.9538, Z -5.5000, A 0.000, B 0.000, C 0.000 }
gfCNCPoint4[6960] = {X 213.3131, Y 51.3749, Z -5.5000, A 0.000, B 0.000, C 0.000 }
gfCNCPoint4[6961] = {X 214.4306, Y 50.9724, Z -5.5000, A 0.000, B 0.000, C 0.000 }
gfCNCPoint4[6962] = {X 215.3724, Y 50.7834, Z -5.5000, A 0.000, B 0.000, C 0.000 }
gfCNCPoint4[6963] = {X 216.3308, Y 50.7200, Z -5.5000, A 0.000, B 0.000, C 0.000 }
gfCNCPoint4[6964] = {X 237.2617, Y 50.7200, Z -5.5000, A 0.000, B 0.000, C 0.000 }
gfCNCPoint4[6965] = {X 238.3057, Y 50.7953, Z -5.5000, A 0.000, B 0.000, C 0.000 }
gfCNCPoint4[6966] = {X 239.3282, Y 51.0195, Z -5.5000, A 0.000, B 0.000, C 0.000 }
gfCNCPoint4[6967] = {X 240.3080, Y 51.3880, Z -5.5000, A 0.000, B 0.000, C 0.000 }
gfCNCPoint4[6968] = {X 241.2247, Y 51.8932, Z -5.5000, A 0.000, B 0.000, C 0.000 }
gfCNCPoint4[6969] = {X 242.0741, Y 52.5375, Z -5.5000, A 0.000, B 0.000, C 0.000 }
gfCNCPoint4[6970] = {X 242.8202, Y 53.2989, Z -5.5000, A 0.000, B 0.000, C 0.000 }
gfCNCPoint4[6971] = {X 243.4472, Y 54.1610, Z -5.5000, A 0.000, B 0.000, C 0.000 }
gfCNCPoint4[6972] = {X 243.9416, Y 55.1055, Z -5.5000, A 0.000, B 0.000, C 0.000 }
gfCNCPoint4[6973] = {X 244.2926, Y 56.1121, Z -5.5000, A 0.000, B 0.000, C 0.000 }
gfCNCPoint4[6974] = {X 249.2037, Y 58.0271, Z -5.5000, A 0.000, B 0.000, C 0.000 }
gfCNCPoint4[6975] = {X 272.6723, Y 67.3422, Z -5.5000, A 0.000, B 0.000, C 0.000 }
gfCNCPoint4[6976] = {X 272.6721, Y 65.2839, Z -5.5000, A 0.000, B 0.000, C 0.000 }
gfCNCPoint4[6977] = {X 271.6647, Y 64.6026, Z -5.5000, A 0.000, B 0.000, C 0.000 }
gfCNCPoint4[6978] = {X 270.7847, Y 63.7630, Z -5.5000, A 0.000, B 0.000, C 0.000 }
gfCNCPoint4[6979] = {X 270.0568, Y 62.7886, Z -5.5000, A 0.000, B 0.000, C 0.000 }
gfCNCPoint4[6980] = {X 269.5013, Y 61.7066, Z -5.5000, A 0.000, B 0.000, C 0.000 }
gfCNCPoint4[6981] = {X 269.2026, Y 60.8252, Z -5.5000, A 0.000, B 0.000, C 0.000 }
gfCNCPoint4[6982] = {X 269.0188, Y 59.9128, Z -5.5000, A 0.000, B 0.000, C 0.000 }
gfCNCPoint4[6983] = {X 268.9529, Y 58.9845, Z -5.5000, A 0.000, B 0.000, C 0.000 }
gfCNCPoint4[6984] = {X 268.9527, Y 58.0000, Z -5.5000, A 0.000, B 0.000, C 0.000 }
gfCNCPoint4[6985] = {X 269.0633, Y 56.7358, Z -5.5000, A 0.000, B 0.000, C 0.000 }
gfCNCPoint4[6986] = {X 269.3917, Y 55.5101, Z -5.5000, A 0.000, B 0.000, C 0.000 }
gfCNCPoint4[6987] = {X 269.9280, Y 54.3600, Z -5.5000, A 0.000, B 0.000, C 0.000 }
gfCNCPoint4[6988] = {X 270.6559, Y 53.3205, Z -5.5000, A 0.000, B 0.000, C 0.000 }
gfCNCPoint4[6989] = {X 271.5532, Y 52.4232, Z -5.5000, A 0.000, B 0.000, C 0.000 }
gfCNCPoint4[6990] = {X 272.5927, Y 51.6953, Z -5.5000, A 0.000, B 0.000, C 0.000 }
gfCNCPoint4[6991] = {X 273.7428, Y 51.1590, Z -5.5000, A 0.000, B 0.000, C 0.000 }
gfCNCPoint4[6992] = {X 274.9685, Y 50.8306, Z -5.5000, A 0.000, B 0.000, C 0.000 }
gfCNCPoint4[6993] = {X 276.2327, Y 50.7200, Z -5.5000, A 0.000, B 0.000, C 0.000 }
gfCNCPoint4[6994] = {X 292.7731, Y 50.7200, Z -5.5000, A 0.000, B 0.000, C 0.000 }
gfCNCPoint4[6995] = {X 293.4209, Y 50.7489, Z -5.5000, A 0.000, B 0.000, C 0.000 }
gfCNCPoint4[6996] = {X 294.0636, Y 50.8353, Z -5.5000, A 0.000, B 0.000, C 0.000 }
gfCNCPoint4[6997] = {X 294.7294, Y 50.9878, Z -5.5000, A 0.000, B 0.000, C 0.000 }
gfCNCPoint4[6998] = {X 295.3779, Y 51.2020, Z -5.5000, A 0.000, B 0.000, C 0.000 }
gfCNCPoint4[6999] = {X 298.3089, Y 43.5526, Z -5.5000, A 0.000, B 0.000, C 0.000 }
gfCNCPoint4[7000] = {X 298.4821, Y 42.5294, Z -5.5000, A 0.000, B 0.000, C 0.000 }
gfCNCPoint4[7001] = {X 298.7925, Y 41.5392, Z -5.5000, A 0.000, B 0.000, C 0.000 }
gfCNCPoint4[7002] = {X 299.2343, Y 40.6002, Z -5.5000, A 0.000, B 0.000, C 0.000 }
gfCNCPoint4[7003] = {X 299.7994, Y 39.7298, Z -5.5000, A 0.000, B 0.000, C 0.000 }
gfCNCPoint4[7004] = {X 299.7994, Y 36.9943, Z -5.5000, A 0.000, B 0.000, C 0.000 }
gfCNCPoint4[7005] = {X 296.8144, Y 36.9943, Z -5.5000, A 0.000, B 0.000, C 0.000 }
gfCNCPoint4[7006] = {X 296.8141, Y 39.7484, Z -5.5000, A 0.000, B 0.000, C 0.000 }
gfCNCPoint4[7007] = {X 297.3853, Y 40.6109, Z -5.5000, A 0.000, B 0.000, C 0.000 }
gfCNCPoint4[7008] = {X 297.8302, Y 41.5449, Z -5.5000, A 0.000, B 0.000, C 0.000 }
gfCNCPoint4[7009] = {X 298.1401, Y 42.5319, Z -5.5000, A 0.000, B 0.000, C 0.000 }
gfCNCPoint4[7010] = {X 298.3089, Y 43.5526, Z -5.5000, A 0.000, B 0.000, C 0.000 }
gfCNCPoint4[7011] = {X 296.2366, Y 48.9608, Z -5.5000, A 0.000, B 0.000, C 0.000 }
gfCNCPoint4[7012] = {X 296.6125, Y 49.1140, Z -5.5000, A 0.000, B 0.000, C 0.000 }
gfCNCPoint4[7013] = {X 296.9817, Y 49.2828, Z -5.5000, A 0.000, B 0.000, C 0.000 }
gfCNCPoint4[7014] = {X 297.2571, Y 49.4212, Z -5.5000, A 0.000, B 0.000, C 0.000 }
gfCNCPoint4[7015] = {X 297.5280, Y 49.5683, Z -5.5000, A 0.000, B 0.000, C 0.000 }
gfCNCPoint4[7016] = {X 298.7174, Y 50.3602, Z -5.5000, A 0.000, B 0.000, C 0.000 }
gfCNCPoint4[7017] = {X 299.7774, Y 51.3185, Z -5.5000, A 0.000, B 0.000, C 0.000 }
gfCNCPoint4[7018] = {X 300.6847, Y 52.4224, Z -5.5000, A 0.000, B 0.000, C 0.000 }
gfCNCPoint4[7019] = {X 301.5914, Y 51.3191, Z -5.5000, A 0.000, B 0.000, C 0.000 }
gfCNCPoint4[7020] = {X 302.6506, Y 50.3611, Z -5.5000, A 0.000, B 0.000, C 0.000 }
gfCNCPoint4[7021] = {X 303.8393, Y 49.5695, Z -5.5000, A 0.000, B 0.000, C 0.000 }
gfCNCPoint4[7022] = {X 302.8989, Y 49.0956, Z -5.5000, A 0.000, B 0.000, C 0.000 }
gfCNCPoint4[7023] = {X 302.0820, Y 48.4310, Z -5.5000, A 0.000, B 0.000, C 0.000 }
gfCNCPoint4[7024] = {X 301.4268, Y 47.6067, Z -5.5000, A 0.000, B 0.000, C 0.000 }
gfCNCPoint4[7025] = {X 300.9636, Y 46.6610, Z -5.5000, A 0.000, B 0.000, C 0.000 }
gfCNCPoint4[7026] = {X 300.7923, Y 46.0759, Z -5.5000, A 0.000, B 0.000, C 0.000 }
gfCNCPoint4[7027] = {X 300.6953, Y 45.4741, Z -5.5000, A 0.000, B 0.000, C 0.000 }
gfCNCPoint4[7028] = {X 300.6790, Y 45.2570, Z -5.5000, A 0.000, B 0.000, C 0.000 }
gfCNCPoint4[7029] = {X 300.6724, Y 45.0393, Z -5.5000, A 0.000, B 0.000, C 0.000 }
gfCNCPoint4[7030] = {X 300.6725, Y 44.1880, Z -5.5000, A 0.000, B 0.000, C 0.000 }
gfCNCPoint4[7031] = {X 300.6810, Y 43.9895, Z -5.5000, A 0.000, B 0.000, C 0.000 }
gfCNCPoint4[7032] = {X 300.6970, Y 43.7913, Z -5.5000, A 0.000, B 0.000, C 0.000 }
gfCNCPoint4[7033] = {X 300.8617, Y 42.9121, Z -5.5000, A 0.000, B 0.000, C 0.000 }
gfCNCPoint4[7034] = {X 301.1738, Y 42.0738, Z -5.5000, A 0.000, B 0.000, C 0.000 }
gfCNCPoint4[7035] = {X 301.6241, Y 41.3009, Z -5.5000, A 0.000, B 0.000, C 0.000 }
gfCNCPoint4[7036] = {X 302.1994, Y 40.6160, Z -5.5000, A 0.000, B 0.000, C 0.000 }
gfCNCPoint4[7037] = {X 302.1994, Y 34.5943, Z -5.5000, A 0.000, B 0.000, C 0.000 }
gfCNCPoint4[7038] = {X 294.4146, Y 34.5943, Z -5.5000, A 0.000, B 0.000, C 0.000 }
gfCNCPoint4[7039] = {X 294.4140, Y 40.6553, Z -5.5000, A 0.000, B 0.000, C 0.000 }
gfCNCPoint4[7040] = {X 294.9942, Y 41.3221, Z -5.5000, A 0.000, B 0.000, C 0.000 }
gfCNCPoint4[7041] = {X 295.4472, Y 42.0809, Z -5.5000, A 0.000, B 0.000, C 0.000 }
gfCNCPoint4[7042] = {X 295.7589, Y 42.9080, Z -5.5000, A 0.000, B 0.000, C 0.000 }
gfCNCPoint4[7043] = {X 295.9194, Y 43.7771, Z -5.5000, A 0.000, B 0.000, C 0.000 }
gfCNCPoint4[7044] = {X 295.9350, Y 43.9928, Z -5.5000, A 0.000, B 0.000, C 0.000 }
gfCNCPoint4[7045] = {X 295.9411, Y 44.2089, Z -5.5000, A 0.000, B 0.000, C 0.000 }
gfCNCPoint4[7046] = {X 295.9411, Y 45.0000, Z -5.5000, A 0.000, B 0.000, C 0.000 }
gfCNCPoint4[7047] = {X 295.9354, Y 45.2373, Z -5.5000, A 0.000, B 0.000, C 0.000 }
gfCNCPoint4[7048] = {X 295.9180, Y 45.4741, Z -5.5000, A 0.000, B 0.000, C 0.000 }
gfCNCPoint4[7049] = {X 298.3067, Y 45.7073, Z -5.5000, A 0.000, B 0.000, C 0.000 }
gfCNCPoint4[7050] = {X 298.2010, Y 46.4214, Z -5.5000, A 0.000, B 0.000, C 0.000 }
gfCNCPoint4[7051] = {X 298.0252, Y 47.1215, Z -5.5000, A 0.000, B 0.000, C 0.000 }
gfCNCPoint4[7052] = {X 298.3689, Y 47.2942, Z -5.5000, A 0.000, B 0.000, C 0.000 }
gfCNCPoint4[7053] = {X 298.7069, Y 47.4778, Z -5.5000, A 0.000, B 0.000, C 0.000 }
gfCNCPoint4[7054] = {X 298.4514, Y 46.6051, Z -5.5000, A 0.000, B 0.000, C 0.000 }
gfCNCPoint4[7055] = {X 298.3067, Y 45.7073, Z -5.5000, A 0.000, B 0.000, C 0.000 }
gfCNCPoint4[7056] = {X 295.9180, Y 45.4741, Z -5.5000, A 0.000, B 0.000, C 0.000 }
gfCNCPoint4[7057] = {X 295.8472, Y 45.9528, Z -5.5000, A 0.000, B 0.000, C 0.000 }
gfCNCPoint4[7058] = {X 295.7293, Y 46.4221, Z -5.5000, A 0.000, B 0.000, C 0.000 }
gfCNCPoint4[7059] = {X 295.4314, Y 47.1714, Z -5.5000, A 0.000, B 0.000, C 0.000 }
gfCNCPoint4[7060] = {X 295.0142, Y 47.8614, Z -5.5000, A 0.000, B 0.000, C 0.000 }
gfCNCPoint4[7061] = {X 294.4890, Y 48.4733, Z -5.5000, A 0.000, B 0.000, C 0.000 }
gfCNCPoint4[7062] = {X 295.3743, Y 48.6760, Z -5.5000, A 0.000, B 0.000, C 0.000 }
gfCNCPoint4[7063] = {X 296.2366, Y 48.9608, Z -5.5000, A 0.000, B 0.000, C 0.000 }
gfCNCPoint4[7064] = {X 295.3779, Y 51.2020, Z -5.5000, A 0.000, B 0.000, C 0.000 }
gfCNCPoint4[7065] = {X 296.3500, Y 51.6593, Z -5.5000, A 0.000, B 0.000, C 0.000 }
gfCNCPoint4[7066] = {X 297.2442, Y 52.2548, Z -5.5000, A 0.000, B 0.000, C 0.000 }
gfCNCPoint4[7067] = {X 298.0410, Y 52.9753, Z -5.5000, A 0.000, B 0.000, C 0.000 }
gfCNCPoint4[7068] = {X 298.7231, Y 53.8053, Z -5.5000, A 0.000, B 0.000, C 0.000 }
gfCNCPoint4[7069] = {X 299.2946, Y 54.7645, Z -5.5000, A 0.000, B 0.000, C 0.000 }
gfCNCPoint4[7070] = {X 299.7126, Y 55.7997, Z -5.5000, A 0.000, B 0.000, C 0.000 }
gfCNCPoint4[7071] = {X 299.9675, Y 56.8868, Z -5.5000, A 0.000, B 0.000, C 0.000 }
gfCNCPoint4[7072] = {X 300.0531, Y 58.0000, Z -5.5000, A 0.000, B 0.000, C 0.000 }
gfCNCPoint4[7073] = {X 300.0531, Y 58.9439, Z -5.5000, A 0.000, B 0.000, C 0.000 }
gfCNCPoint4[7074] = {X 299.9648, Y 60.0538, Z -5.5000, A 0.000, B 0.000, C 0.000 }
gfCNCPoint4[7075] = {X 299.7087, Y 61.1373, Z -5.5000, A 0.000, B 0.000, C 0.000 }
gfCNCPoint4[7076] = {X 299.2907, Y 62.1692, Z -5.5000, A 0.000, B 0.000, C 0.000 }
gfCNCPoint4[7077] = {X 298.7206, Y 63.1256, Z -5.5000, A 0.000, B 0.000, C 0.000 }
gfCNCPoint4[7078] = {X 300.6823, Y 64.5083, Z -5.5000, A 0.000, B 0.000, C 0.000 }
gfCNCPoint4[7079] = {X 299.7828, Y 65.6044, Z -5.5000, A 0.000, B 0.000, C 0.000 }
gfCNCPoint4[7080] = {X 298.7331, Y 66.5577, Z -5.5000, A 0.000, B 0.000, C 0.000 }
gfCNCPoint4[7081] = {X 298.7331, Y 89.4419, Z -5.5000, A 0.000, B 0.000, C 0.000 }
gfCNCPoint4[7082] = {X 299.8298, Y 90.4464, Z -5.5000, A 0.000, B 0.000, C 0.000 }
gfCNCPoint4[7083] = {X 300.7602, Y 91.6065, Z -5.5000, A 0.000, B 0.000, C 0.000 }
gfCNCPoint4[7084] = {X 301.5027, Y 92.8951, Z -5.5000, A 0.000, B 0.000, C 0.000 }
gfCNCPoint4[7085] = {X 304.0670, Y 92.8951, Z -5.5000, A 0.000, B 0.000, C 0.000 }
gfCNCPoint4[7086] = {X 303.7095, Y 91.9004, Z -5.5000, A 0.000, B 0.000, C 0.000 }
gfCNCPoint4[7087] = {X 303.4134, Y 90.8857, Z -5.5000, A 0.000, B 0.000, C 0.000 }
gfCNCPoint4[7088] = {X 302.9742, Y 88.8149, Z -5.5000, A 0.000, B 0.000, C 0.000 }
gfCNCPoint4[7089] = {X 302.7141, Y 86.7142, Z -5.5000, A 0.000, B 0.000, C 0.000 }
gfCNCPoint4[7090] = {X 302.6350, Y 84.5988, Z -5.5000, A 0.000, B 0.000, C 0.000 }
gfCNCPoint4[7091] = {X 302.6361, Y 66.5616, Z -5.5000, A 0.000, B 0.000, C 0.000 }
gfCNCPoint4[7092] = {X 301.5836, Y 65.6068, Z -5.5000, A 0.000, B 0.000, C 0.000 }
gfCNCPoint4[7093] = {X 300.6823, Y 64.5083, Z -5.5000, A 0.000, B 0.000, C 0.000 }
gfCNCPoint4[7094] = {X 298.7206, Y 63.1256, Z -5.5000, A 0.000, B 0.000, C 0.000 }
gfCNCPoint4[7095] = {X 298.0346, Y 63.9600, Z -5.5000, A 0.000, B 0.000, C 0.000 }
gfCNCPoint4[7096] = {X 297.2329, Y 64.6841, Z -5.5000, A 0.000, B 0.000, C 0.000 }
gfCNCPoint4[7097] = {X 296.3331, Y 65.2818, Z -5.5000, A 0.000, B 0.000, C 0.000 }
gfCNCPoint4[7098] = {X 296.3331, Y 90.7162, Z -5.5000, A 0.000, B 0.000, C 0.000 }
gfCNCPoint4[7099] = {X 297.3132, Y 91.3790, Z -5.5000, A 0.000, B 0.000, C 0.000 }
gfCNCPoint4[7100] = {X 298.1737, Y 92.1911, Z -5.5000, A 0.000, B 0.000, C 0.000 }
gfCNCPoint4[7101] = {X 298.8919, Y 93.1313, Z -5.5000, A 0.000, B 0.000, C 0.000 }
gfCNCPoint4[7102] = {X 299.4490, Y 94.1751, Z -5.5000, A 0.000, B 0.000, C 0.000 }
gfCNCPoint4[7103] = {X 299.8306, Y 95.2951, Z -5.5000, A 0.000, B 0.000, C 0.000 }
gfCNCPoint4[7104] = {X 308.0990, Y 95.2951, Z -5.5000, A 0.000, B 0.000, C 0.000 }
gfCNCPoint4[7105] = {X 307.0958, Y 93.7116, Z -5.5000, A 0.000, B 0.000, C 0.000 }
gfCNCPoint4[7106] = {X 306.2996, Y 92.0145, Z -5.5000, A 0.000, B 0.000, C 0.000 }
gfCNCPoint4[7107] = {X 305.9917, Y 91.1580, Z -5.5000, A 0.000, B 0.000, C 0.000 }
gfCNCPoint4[7108] = {X 305.7368, Y 90.2842, Z -5.5000, A 0.000, B 0.000, C 0.000 }
gfCNCPoint4[7109] = {X 305.3405, Y 88.4138, Z -5.5000, A 0.000, B 0.000, C 0.000 }
gfCNCPoint4[7110] = {X 305.1060, Y 86.5163, Z -5.5000, A 0.000, B 0.000, C 0.000 }
gfCNCPoint4[7111] = {X 305.0350, Y 84.6058, Z -5.5000, A 0.000, B 0.000, C 0.000 }
gfCNCPoint4[7112] = {X 305.0362, Y 65.2842, Z -5.5000, A 0.000, B 0.000, C 0.000 }
gfCNCPoint4[7113] = {X 304.1345, Y 64.6866, Z -5.5000, A 0.000, B 0.000, C 0.000 }
gfCNCPoint4[7114] = {X 303.3313, Y 63.9619, Z -5.5000, A 0.000, B 0.000, C 0.000 }
gfCNCPoint4[7115] = {X 302.6444, Y 63.1262, Z -5.5000, A 0.000, B 0.000, C 0.000 }
gfCNCPoint4[7116] = {X 302.0793, Y 62.1788, Z -5.5000, A 0.000, B 0.000, C 0.000 }
gfCNCPoint4[7117] = {X 301.6639, Y 61.1568, Z -5.5000, A 0.000, B 0.000, C 0.000 }
gfCNCPoint4[7118] = {X 301.4076, Y 60.0839, Z -5.5000, A 0.000, B 0.000, C 0.000 }
gfCNCPoint4[7119] = {X 301.3164, Y 58.9845, Z -5.5000, A 0.000, B 0.000, C 0.000 }
gfCNCPoint4[7120] = {X 301.3162, Y 58.0000, Z -5.5000, A 0.000, B 0.000, C 0.000 }
gfCNCPoint4[7121] = {X 301.4018, Y 56.8868, Z -5.5000, A 0.000, B 0.000, C 0.000 }
gfCNCPoint4[7122] = {X 301.6567, Y 55.7997, Z -5.5000, A 0.000, B 0.000, C 0.000 }
gfCNCPoint4[7123] = {X 302.0747, Y 54.7645, Z -5.5000, A 0.000, B 0.000, C 0.000 }
gfCNCPoint4[7124] = {X 302.6462, Y 53.8053, Z -5.5000, A 0.000, B 0.000, C 0.000 }
gfCNCPoint4[7125] = {X 303.3281, Y 52.9755, Z -5.5000, A 0.000, B 0.000, C 0.000 }
gfCNCPoint4[7126] = {X 304.1247, Y 52.2551, Z -5.5000, A 0.000, B 0.000, C 0.000 }
gfCNCPoint4[7127] = {X 305.0187, Y 51.6597, Z -5.5000, A 0.000, B 0.000, C 0.000 }
gfCNCPoint4[7128] = {X 306.1514, Y 51.1428, Z -5.5000, A 0.000, B 0.000, C 0.000 }
gfCNCPoint4[7129] = {X 307.3557, Y 50.8265, Z -5.5000, A 0.000, B 0.000, C 0.000 }
gfCNCPoint4[7130] = {X 308.5962, Y 50.7200, Z -5.5000, A 0.000, B 0.000, C 0.000 }
gfCNCPoint4[7131] = {X 324.3107, Y 50.7200, Z -5.5000, A 0.000, B 0.000, C 0.000 }
gfCNCPoint4[7132] = {X 325.2469, Y 50.7804, Z -5.5000, A 0.000, B 0.000, C 0.000 }
gfCNCPoint4[7133] = {X 326.1675, Y 50.9608, Z -5.5000, A 0.000, B 0.000, C 0.000 }
gfCNCPoint4[7134] = {X 326.5260, Y 51.0653, Z -5.5000, A 0.000, B 0.000, C 0.000 }
gfCNCPoint4[7135] = {X 326.8787, Y 51.1880, Z -5.5000, A 0.000, B 0.000, C 0.000 }
gfCNCPoint4[7136] = {X 327.4493, Y 51.4313, Z -5.5000, A 0.000, B 0.000, C 0.000 }
gfCNCPoint4[7137] = {X 327.9972, Y 51.7224, Z -5.5000, A 0.000, B 0.000, C 0.000 }
gfCNCPoint4[7138] = {X 328.5425, Y 52.0763, Z -5.5000, A 0.000, B 0.000, C 0.000 }
gfCNCPoint4[7139] = {X 329.0541, Y 52.4775, Z -5.5000, A 0.000, B 0.000, C 0.000 }
gfCNCPoint4[7140] = {X 329.9304, Y 53.3721, Z -5.5000, A 0.000, B 0.000, C 0.000 }
gfCNCPoint4[7141] = {X 330.6404, Y 54.4037, Z -5.5000, A 0.000, B 0.000, C 0.000 }
gfCNCPoint4[7142] = {X 331.1630, Y 55.5416, Z -5.5000, A 0.000, B 0.000, C 0.000 }
gfCNCPoint4[7143] = {X 331.4830, Y 56.7524, Z -5.5000, A 0.000, B 0.000, C 0.000 }
gfCNCPoint4[7144] = {X 331.5907, Y 58.0000, Z -5.5000, A 0.000, B 0.000, C 0.000 }
gfCNCPoint4[7145] = {X 331.5907, Y 58.9396, Z -5.5000, A 0.000, B 0.000, C 0.000 }
gfCNCPoint4[7146] = {X 331.4734, Y 60.2166, Z -5.5000, A 0.000, B 0.000, C 0.000 }
gfCNCPoint4[7147] = {X 331.1351, Y 61.4536, Z -5.5000, A 0.000, B 0.000, C 0.000 }
gfCNCPoint4[7148] = {X 330.5860, Y 62.6124, Z -5.5000, A 0.000, B 0.000, C 0.000 }
gfCNCPoint4[7149] = {X 329.8430, Y 63.6577, Z -5.5000, A 0.000, B 0.000, C 0.000 }
gfCNCPoint4[7150] = {X 328.9290, Y 64.5572, Z -5.5000, A 0.000, B 0.000, C 0.000 }
gfCNCPoint4[7151] = {X 327.8720, Y 65.2833, Z -5.5000, A 0.000, B 0.000, C 0.000 }
gfCNCPoint4[7152] = {X 327.8736, Y 83.2150, Z -5.5000, A 0.000, B 0.000, C 0.000 }
gfCNCPoint4[7153] = {X 327.8870, Y 84.5915, Z -5.5000, A 0.000, B 0.000, C 0.000 }
gfCNCPoint4[7154] = {X 327.8966, Y 84.9540, Z -5.5000, A 0.000, B 0.000, C 0.000 }
gfCNCPoint4[7155] = {X 327.9234, Y 85.3157, Z -5.5000, A 0.000, B 0.000, C 0.000 }
gfCNCPoint4[7156] = {X 328.8617, Y 85.6718, Z -5.5000, A 0.000, B 0.000, C 0.000 }
gfCNCPoint4[7157] = {X 329.8280, Y 85.9428, Z -5.5000, A 0.000, B 0.000, C 0.000 }
gfCNCPoint4[7158] = {X 331.9609, Y 86.3869, Z -5.5000, A 0.000, B 0.000, C 0.000 }
gfCNCPoint4[7159] = {X 334.1130, Y 86.7257, Z -5.5000, A 0.000, B 0.000, C 0.000 }
gfCNCPoint4[7160] = {X 336.2791, Y 86.9583, Z -5.5000, A 0.000, B 0.000, C 0.000 }
gfCNCPoint4[7161] = {X 340.5610, Y 87.2466, Z -5.5000, A 0.000, B 0.000, C 0.000 }
gfCNCPoint4[7162] = {X 344.8499, Y 87.3971, Z -5.5000, A 0.000, B 0.000, C 0.000 }
gfCNCPoint4[7163] = {X 349.1414, Y 87.4097, Z -5.5000, A 0.000, B 0.000, C 0.000 }
gfCNCPoint4[7164] = {X 353.1932, Y 87.3438, Z -5.5000, A 0.000, B 0.000, C 0.000 }
gfCNCPoint4[7165] = {X 357.2400, Y 87.1306, Z -5.5000, A 0.000, B 0.000, C 0.000 }
gfCNCPoint4[7166] = {X 361.2763, Y 86.7704, Z -5.5000, A 0.000, B 0.000, C 0.000 }
gfCNCPoint4[7167] = {X 363.1972, Y 86.5052, Z -5.5000, A 0.000, B 0.000, C 0.000 }
gfCNCPoint4[7168] = {X 365.1003, Y 86.1338, Z -5.5000, A 0.000, B 0.000, C 0.000 }
gfCNCPoint4[7169] = {X 366.9800, Y 85.6574, Z -5.5000, A 0.000, B 0.000, C 0.000 }
gfCNCPoint4[7170] = {X 367.4412, Y 85.5109, Z -5.5000, A 0.000, B 0.000, C 0.000 }
gfCNCPoint4[7171] = {X 367.8885, Y 85.3264, Z -5.5000, A 0.000, B 0.000, C 0.000 }
gfCNCPoint4[7172] = {X 367.9420, Y 84.5784, Z -5.5000, A 0.000, B 0.000, C 0.000 }
gfCNCPoint4[7173] = {X 367.9597, Y 83.8287, Z -5.5000, A 0.000, B 0.000, C 0.000 }
gfCNCPoint4[7174] = {X 367.9585, Y 65.2838, Z -5.5000, A 0.000, B 0.000, C 0.000 }
gfCNCPoint4[7175] = {X 366.9047, Y 64.5647, Z -5.5000, A 0.000, B 0.000, C 0.000 }
gfCNCPoint4[7176] = {X 365.9927, Y 63.6727, Z -5.5000, A 0.000, B 0.000, C 0.000 }
gfCNCPoint4[7177] = {X 365.2503, Y 62.6352, Z -5.5000, A 0.000, B 0.000, C 0.000 }
gfCNCPoint4[7178] = {X 364.7005, Y 61.4840, Z -5.5000, A 0.000, B 0.000, C 0.000 }
gfCNCPoint4[7179] = {X 364.3600, Y 60.2545, Z -5.5000, A 0.000, B 0.000, C 0.000 }
gfCNCPoint4[7180] = {X 364.2395, Y 58.9845, Z -5.5000, A 0.000, B 0.000, C 0.000 }
gfCNCPoint4[7181] = {X 364.2393, Y 58.0000, Z -5.5000, A 0.000, B 0.000, C 0.000 }
gfCNCPoint4[7182] = {X 364.3499, Y 56.7358, Z -5.5000, A 0.000, B 0.000, C 0.000 }
gfCNCPoint4[7183] = {X 364.6783, Y 55.5101, Z -5.5000, A 0.000, B 0.000, C 0.000 }
gfCNCPoint4[7184] = {X 365.2146, Y 54.3600, Z -5.5000, A 0.000, B 0.000, C 0.000 }
gfCNCPoint4[7185] = {X 365.9425, Y 53.3205, Z -5.5000, A 0.000, B 0.000, C 0.000 }
gfCNCPoint4[7186] = {X 366.8398, Y 52.4232, Z -5.5000, A 0.000, B 0.000, C 0.000 }
gfCNCPoint4[7187] = {X 367.8793, Y 51.6953, Z -5.5000, A 0.000, B 0.000, C 0.000 }
gfCNCPoint4[7188] = {X 369.0294, Y 51.1590, Z -5.5000, A 0.000, B 0.000, C 0.000 }
gfCNCPoint4[7189] = {X 370.2551, Y 50.8306, Z -5.5000, A 0.000, B 0.000, C 0.000 }
gfCNCPoint4[7190] = {X 371.5193, Y 50.7200, Z -5.5000, A 0.000, B 0.000, C 0.000 }
gfCNCPoint4[7191] = {X 388.0597, Y 50.7200, Z -5.5000, A 0.000, B 0.000, C 0.000 }
gfCNCPoint4[7192] = {X 389.2271, Y 50.8142, Z -5.5000, A 0.000, B 0.000, C 0.000 }
gfCNCPoint4[7193] = {X 390.3643, Y 51.0944, Z -5.5000, A 0.000, B 0.000, C 0.000 }
gfCNCPoint4[7194] = {X 391.4418, Y 51.5533, Z -5.5000, A 0.000, B 0.000, C 0.000 }
gfCNCPoint4[7195] = {X 392.4319, Y 52.1791, Z -5.5000, A 0.000, B 0.000, C 0.000 }
gfCNCPoint4[7196] = {X 393.3087, Y 52.9556, Z -5.5000, A 0.000, B 0.000, C 0.000 }
gfCNCPoint4[7197] = {X 394.1855, Y 52.1791, Z -5.5000, A 0.000, B 0.000, C 0.000 }
gfCNCPoint4[7198] = {X 395.1756, Y 51.5533, Z -5.5000, A 0.000, B 0.000, C 0.000 }
gfCNCPoint4[7199] = {X 396.2531, Y 51.0944, Z -5.5000, A 0.000, B 0.000, C 0.000 }
gfCNCPoint4[7200] = {X 397.3903, Y 50.8142, Z -5.5000, A 0.000, B 0.000, C 0.000 }
gfCNCPoint4[7201] = {X 398.5577, Y 50.7200, Z -5.5000, A 0.000, B 0.000, C 0.000 }
gfCNCPoint4[7202] = {X 419.4886, Y 50.7200, Z -5.5000, A 0.000, B 0.000, C 0.000 }
gfCNCPoint4[7203] = {X 420.6739, Y 50.8171, Z -5.5000, A 0.000, B 0.000, C 0.000 }
gfCNCPoint4[7204] = {X 421.8276, Y 51.1060, Z -5.5000, A 0.000, B 0.000, C 0.000 }
gfCNCPoint4[7205] = {X 422.9189, Y 51.5788, Z -5.5000, A 0.000, B 0.000, C 0.000 }
gfCNCPoint4[7206] = {X 423.9186, Y 52.2230, Z -5.5000, A 0.000, B 0.000, C 0.000 }
gfCNCPoint4[7207] = {X 424.8001, Y 53.0214, Z -5.5000, A 0.000, B 0.000, C 0.000 }
gfCNCPoint4[7208] = {X 425.5398, Y 53.9526, Z -5.5000, A 0.000, B 0.000, C 0.000 }
gfCNCPoint4[7209] = {X 426.1181, Y 54.9919, Z -5.5000, A 0.000, B 0.000, C 0.000 }
gfCNCPoint4[7210] = {X 426.5194, Y 56.1114, Z -5.5000, A 0.000, B 0.000, C 0.000 }
gfCNCPoint4[7211] = {X 430.7006, Y 57.7406, Z -5.5000, A 0.000, B 0.000, C 0.000 }
gfCNCPoint4[7212] = {X 454.8986, Y 67.3415, Z -5.5000, A 0.000, B 0.000, C 0.000 }
gfCNCPoint4[7213] = {X 454.8987, Y 65.2837, Z -5.5000, A 0.000, B 0.000, C 0.000 }
gfCNCPoint4[7214] = {X 453.8915, Y 64.6024, Z -5.5000, A 0.000, B 0.000, C 0.000 }
gfCNCPoint4[7215] = {X 453.0117, Y 63.7630, Z -5.5000, A 0.000, B 0.000, C 0.000 }
gfCNCPoint4[7216] = {X 452.2839, Y 62.7888, Z -5.5000, A 0.000, B 0.000, C 0.000 }
gfCNCPoint4[7217] = {X 451.7284, Y 61.7071, Z -5.5000, A 0.000, B 0.000, C 0.000 }
gfCNCPoint4[7218] = {X 451.4296, Y 60.8255, Z -5.5000, A 0.000, B 0.000, C 0.000 }
gfCNCPoint4[7219] = {X 451.2457, Y 59.9130, Z -5.5000, A 0.000, B 0.000, C 0.000 }
gfCNCPoint4[7220] = {X 451.1798, Y 58.9845, Z -5.5000, A 0.000, B 0.000, C 0.000 }
gfCNCPoint4[7221] = {X 451.1796, Y 58.0000, Z -5.5000, A 0.000, B 0.000, C 0.000 }
gfCNCPoint4[7222] = {X 451.2795, Y 56.7981, Z -5.5000, A 0.000, B 0.000, C 0.000 }
gfCNCPoint4[7223] = {X 451.5765, Y 55.6291, Z -5.5000, A 0.000, B 0.000, C 0.000 }
gfCNCPoint4[7224] = {X 452.0624, Y 54.5253, Z -5.5000, A 0.000, B 0.000, C 0.000 }
gfCNCPoint4[7225] = {X 452.7238, Y 53.5168, Z -5.5000, A 0.000, B 0.000, C 0.000 }
gfCNCPoint4[7226] = {X 453.5427, Y 52.6313, Z -5.5000, A 0.000, B 0.000, C 0.000 }
gfCNCPoint4[7227] = {X 454.4966, Y 51.8932, Z -5.5000, A 0.000, B 0.000, C 0.000 }
gfCNCPoint4[7228] = {X 455.4133, Y 51.3880, Z -5.5000, A 0.000, B 0.000, C 0.000 }
gfCNCPoint4[7229] = {X 456.3931, Y 51.0195, Z -5.5000, A 0.000, B 0.000, C 0.000 }
gfCNCPoint4[7230] = {X 457.4155, Y 50.7953, Z -5.5000, A 0.000, B 0.000, C 0.000 }
gfCNCPoint4[7231] = {X 458.4596, Y 50.7200, Z -5.5000, A 0.000, B 0.000, C 0.000 }
gfCNCPoint4[7232] = {X 475.0000, Y 50.7200, Z -5.5000, A 0.000, B 0.000, C 0.000 }
gfCNCPoint4[7233] = {X 476.0441, Y 50.7953, Z -5.5000, A 0.000, B 0.000, C 0.000 }
gfCNCPoint4[7234] = {X 477.0665, Y 51.0195, Z -5.5000, A 0.000, B 0.000, C 0.000 }
gfCNCPoint4[7235] = {X 478.0463, Y 51.3880, Z -5.5000, A 0.000, B 0.000, C 0.000 }
gfCNCPoint4[7236] = {X 478.9630, Y 51.8932, Z -5.5000, A 0.000, B 0.000, C 0.000 }
gfCNCPoint4[7237] = {X 479.9169, Y 52.6313, Z -5.5000, A 0.000, B 0.000, C 0.000 }
gfCNCPoint4[7238] = {X 480.7358, Y 53.5168, Z -5.5000, A 0.000, B 0.000, C 0.000 }
gfCNCPoint4[7239] = {X 481.3972, Y 54.5253, Z -5.5000, A 0.000, B 0.000, C 0.000 }
gfCNCPoint4[7240] = {X 481.8831, Y 55.6291, Z -5.5000, A 0.000, B 0.000, C 0.000 }
gfCNCPoint4[7241] = {X 482.1801, Y 56.7981, Z -5.5000, A 0.000, B 0.000, C 0.000 }
gfCNCPoint4[7242] = {X 482.2800, Y 58.0000, Z -5.5000, A 0.000, B 0.000, C 0.000 }
gfCNCPoint4[7243] = {X 482.2798, Y 58.9942, Z -5.5000, A 0.000, B 0.000, C 0.000 }
gfCNCPoint4[7244] = {X 482.1578, Y 60.2625, Z -5.5000, A 0.000, B 0.000, C 0.000 }
gfCNCPoint4[7245] = {X 481.8165, Y 61.4902, Z -5.5000, A 0.000, B 0.000, C 0.000 }
gfCNCPoint4[7246] = {X 481.2664, Y 62.6395, Z -5.5000, A 0.000, B 0.000, C 0.000 }
gfCNCPoint4[7247] = {X 480.5244, Y 63.6753, Z -5.5000, A 0.000, B 0.000, C 0.000 }
gfCNCPoint4[7248] = {X 479.6131, Y 64.5659, Z -5.5000, A 0.000, B 0.000, C 0.000 }
gfCNCPoint4[7249] = {X 478.5605, Y 65.2840, Z -5.5000, A 0.000, B 0.000, C 0.000 }
gfCNCPoint4[7250] = {X 478.5609, Y 90.7240, Z -5.5000, A 0.000, B 0.000, C 0.000 }
gfCNCPoint4[7251] = {X 479.5435, Y 91.3827, Z -5.5000, A 0.000, B 0.000, C 0.000 }
gfCNCPoint4[7252] = {X 480.4060, Y 92.1923, Z -5.5000, A 0.000, B 0.000, C 0.000 }
gfCNCPoint4[7253] = {X 481.1253, Y 93.1313, Z -5.5000, A 0.000, B 0.000, C 0.000 }
gfCNCPoint4[7254] = {X 481.6825, Y 94.1749, Z -5.5000, A 0.000, B 0.000, C 0.000 }
gfCNCPoint4[7255] = {X 482.0626, Y 95.2951, Z -5.5000, A 0.000, B 0.000, C 0.000 }
gfCNCPoint4[7256] = {X 507.6814, Y 95.2951, Z -5.5000, A 0.000, B 0.000, C 0.000 }
gfCNCPoint4[7257] = {X 507.6814, Y 97.6951, Z -5.5000, A 0.000, B 0.000, C 0.000 }
gfCNCPoint4[7258] = {X 597.6966, Y 97.6951, Z -5.5000, A 0.000, B 0.000, C 0.000 }
gfCNCPoint4[7259] = {X 597.6966, Y 51.8000, Z -5.5000, A 0.000, B 0.000, C 0.000 }
gfCNCPoint4[7260] = {X 593.5565, Y 51.8000, Z -5.5000, A 0.000, B 0.000, C 0.000 }
gfCNCPoint4[7261] = {X 592.3428, Y 51.6908, Z -5.5000, A 0.000, B 0.000, C 0.000 }
gfCNCPoint4[7262] = {X 591.1680, Y 51.3667, Z -5.5000, A 0.000, B 0.000, C 0.000 }
gfCNCPoint4[7263] = {X 590.0699, Y 50.8381, Z -5.5000, A 0.000, B 0.000, C 0.000 }
gfCNCPoint4[7264] = {X 589.0838, Y 50.1220, Z -5.5000, A 0.000, B 0.000, C 0.000 }
gfCNCPoint4[7265] = {X 588.4736, Y 49.5171, Z -5.5000, A 0.000, B 0.000, C 0.000 }
gfCNCPoint4[7266] = {X 587.9446, Y 48.8401, Z -5.5000, A 0.000, B 0.000, C 0.000 }
